Yaskawa INFORM job: tourneTRJ3.JBI

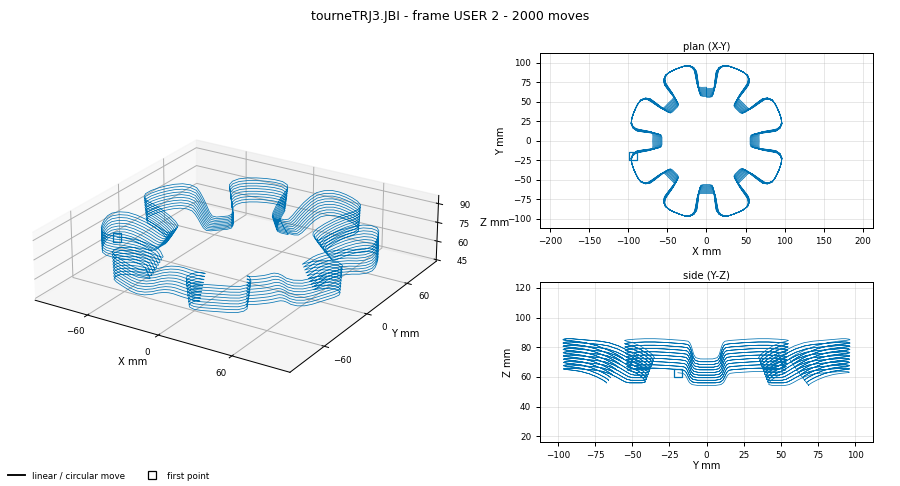
[picture p0: tool path of tourneTRJ3.JBI in frame USER 2, 2000 of 2000 moves have a stored position in this frame; points joined in program order, loops and branches not executed]
/JOB
//NAME tourneTRJ3
///FOLDERNAME DEMO
//POS
///NPOS 2000,0,2000,0,0,0
///USER 2
///TOOL 7
///POSTYPE USER
///RECTAN
///RCONF 1,0,0,0,0,0,0,0,0,0,0,0,0,0,0,0,0,0,0,0,0,0,0,0
C00000=-94.423,-19.246,62.877,176.4713,-3.4802,-10698.4794
C00001=-90.636,-15.942,62.469,177.8869,-7.7734,-10700.0243
C00002=-85.405,-14.621,61.698,179.5492,-7.9435,-10700.2854
C00003=-79.780,-13.569,60.151,179.7039,-6.1061,-10700.3475
C00004=-74.809,-12.586,58.158,179.7463,-3.0888,-10700.4499
C00005=-71.127,-11.507,56.252,-179.3006,3.5805,-10700.8103
C00006=-69.044,-9.699,54.888,-155.7698,19.6431,-10702.0037
C00007=-68.619,-6.200,54.350,-141.8645,5.1067,-10704.8371
C00008=-68.781,-2.945,54.326,-141.2129,-0.2944,-10707.5483
C00009=-68.843,0.000,54.342,-141.2230,0.0000,-10710.0000
C00010=-68.781,2.945,54.326,-141.2129,0.2944,-10712.4517
C00011=-68.619,6.200,54.350,-141.8645,-5.1067,-10715.1629
C00012=-69.044,9.699,54.888,-155.7643,-19.6439,-10717.9963
C00013=-71.127,11.507,56.252,-179.3006,-3.5805,-10719.1897
C00014=-74.809,12.586,58.158,179.7463,3.0888,-10719.5501
C00015=-79.780,13.569,60.151,179.7039,6.1061,-10719.6525
C00016=-85.405,14.621,61.698,179.5492,7.9435,-10719.7146
C00017=-90.636,15.942,62.469,177.8869,7.7734,-10719.9757
C00018=-94.423,19.246,62.877,176.4713,3.4802,-10721.5206
C00019=-96.154,24.159,63.210,177.6712,0.8456,-10724.1038
C00020=-95.429,29.718,63.547,179.8441,0.0005,-10727.2974
C00021=-93.512,35.416,63.770,179.9819,0.0007,-10730.7433
C00022=-91.166,41.080,63.770,179.9820,0.0018,-10734.2566
C00023=-88.493,46.465,63.547,179.8436,-0.0020,-10737.7026
C00024=-85.074,50.908,63.210,177.6714,-0.8446,-10740.8962
C00025=-80.376,53.158,62.877,176.4684,-3.4763,-10743.4793
C00026=-75.362,52.817,62.469,177.8861,-7.7686,-10745.0245
C00027=-70.729,50.052,61.698,179.5510,-7.9442,-10745.2855
C00028=-66.007,46.818,60.151,179.7042,-6.1110,-10745.3476
C00029=-61.798,43.998,58.158,179.7506,-3.0878,-10745.4495
C00030=-58.431,42.158,56.252,-179.3002,3.5752,-10745.8105
C00031=-55.679,41.963,54.888,-155.7662,19.6450,-10747.0038
C00032=-52.905,44.137,54.350,-141.8624,5.1087,-10749.8372
C00033=-50.718,46.553,54.326,-141.2122,-0.2913,-10752.5482
C00034=-48.679,48.679,54.342,-141.2237,-0.0052,-10755.0000
C00035=-46.553,50.718,54.326,-141.2122,0.2913,-10757.4518
C00036=-44.137,52.905,54.350,-141.8624,-5.1087,-10760.1628
C00037=-41.963,55.680,54.888,-155.7664,-19.6452,-10762.9966
C00038=-42.158,58.431,56.252,-179.3002,-3.5752,-10764.1895
C00039=-43.998,61.798,58.158,179.7506,3.0878,-10764.5505
C00040=-46.818,66.007,60.151,179.7042,6.1110,-10764.6524
C00041=-50.052,70.729,61.698,179.5510,7.9442,-10764.7145
C00042=-52.817,75.362,62.469,177.8861,7.7686,-10764.9755
C00043=-53.158,80.376,62.877,176.4684,3.4763,-10766.5207
C00044=-50.908,85.074,63.210,177.6714,0.8446,-10769.1038
C00045=-46.465,88.493,63.547,179.8436,0.0020,-10772.2974
C00046=-41.080,91.166,63.770,179.9820,-0.0018,-10775.7434
C00047=-35.416,93.512,63.770,179.9819,-0.0007,-10779.2567
C00048=-29.718,95.429,63.547,179.8441,-0.0005,-10782.7026
C00049=-24.159,96.154,63.210,177.6712,-0.8456,-10785.8962
C00050=-19.246,94.423,62.877,176.4713,-3.4802,-10788.4794
C00051=-15.942,90.636,62.469,177.8869,-7.7734,-10790.0243
C00052=-14.621,85.405,61.698,179.5492,-7.9435,-10790.2854
C00053=-13.569,79.780,60.151,179.7039,-6.1061,-10790.3475
C00054=-12.586,74.809,58.158,179.7463,-3.0888,-10790.4499
C00055=-11.507,71.127,56.252,-179.3006,3.5805,-10790.8103
C00056=-9.699,69.044,54.888,-155.7643,19.6439,-10792.0037
C00057=-6.200,68.619,54.350,-141.8645,5.1067,-10794.8371
C00058=-2.945,68.781,54.326,-141.2129,-0.2944,-10797.5483
C00059=0.000,68.843,54.342,-141.2230,-0.0000,-10800.0000
C00060=0.000,67.469,56.061,-141.5406,-0.0000,-10800.0000
C00061=2.820,67.413,56.044,-141.5283,0.3002,-10802.3954
C00062=5.989,67.263,56.069,-142.2439,-5.3506,-10805.0881
C00063=9.441,67.734,56.637,-157.1153,-19.5601,-10807.9350
C00064=11.191,69.937,58.076,-179.5522,-2.6083,-10809.0911
C00065=12.227,73.809,60.085,179.7607,3.4681,-10809.4060
C00066=13.183,79.025,62.181,179.7489,6.2113,-10809.4709
C00067=14.211,84.918,63.804,179.6316,7.9111,-10809.5004
C00068=15.500,90.396,64.610,178.0217,7.7526,-10809.7298
C00069=18.832,94.373,65.037,176.5110,3.5309,-10811.2851
C00070=23.832,96.213,65.385,177.6850,0.8573,-10813.9122
C00071=29.513,95.497,65.736,179.8387,0.0019,-10817.1736
C00072=35.347,93.539,65.969,179.9819,0.0007,-10820.7008
C00073=41.148,91.136,65.969,179.9820,0.0019,-10824.2992
C00074=46.658,88.395,65.736,179.8436,-0.0017,-10827.8267
C00075=51.181,84.885,65.385,177.6852,-0.8535,-10831.0877
C00076=53.416,80.048,65.037,176.5097,-3.5333,-10833.7152
C00077=52.959,74.880,64.610,178.0182,-7.7554,-10835.2699
C00078=49.997,70.095,63.804,179.6281,-7.9119,-10835.4993
C00079=46.557,65.200,62.181,179.7470,-6.2113,-10835.5293
C00080=43.545,60.837,60.085,179.7604,-3.4666,-10835.5938
C00081=41.540,57.367,58.076,-179.5517,2.6125,-10835.9087
C00082=41.220,54.571,56.637,-157.1158,19.5601,-10837.0654
C00083=43.327,51.796,56.069,-142.2456,5.3482,-10839.9123
C00084=45.674,49.662,56.044,-141.5313,-0.2969,-10842.6047
C00085=47.708,47.708,56.061,-141.5419,-0.0000,-10845.0000
C00086=49.662,45.674,56.044,-141.5313,0.2969,-10847.3953
C00087=51.797,43.327,56.069,-142.2457,-5.3486,-10850.0883
C00088=54.571,41.220,56.637,-157.1158,-19.5601,-10852.9346
C00089=57.367,41.540,58.076,-179.5517,-2.6125,-10854.0913
C00090=60.837,43.545,60.085,179.7604,3.4666,-10854.4062
C00091=65.200,46.557,62.181,179.7470,6.2113,-10854.4707
C00092=70.095,49.997,63.804,179.6281,7.9119,-10854.5007
C00093=74.880,52.959,64.610,178.0182,7.7554,-10854.7301
C00094=80.048,53.416,65.037,176.5097,3.5333,-10856.2848
C00095=84.885,51.181,65.385,177.6852,0.8535,-10858.9123
C00096=88.395,46.658,65.736,179.8436,0.0017,-10862.1733
C00097=91.136,41.148,65.969,179.9820,-0.0019,-10865.7008
C00098=93.539,35.347,65.969,179.9819,-0.0007,-10869.2992
C00099=95.497,29.513,65.736,179.8387,-0.0019,-10872.8264
C00100=96.213,23.832,65.385,177.6850,-0.8573,-10876.0878
C00101=94.373,18.832,65.037,176.5110,-3.5309,-10878.7149
C00102=90.396,15.500,64.610,178.0217,-7.7526,-10880.2702
C00103=84.918,14.211,63.804,179.6316,-7.9111,-10880.4996
C00104=79.025,13.183,62.181,179.7489,-6.2113,-10880.5291
C00105=73.809,12.227,60.085,179.7607,-3.4681,-10880.5940
C00106=69.937,11.191,58.076,-179.5522,2.6083,-10880.9089
C00107=67.734,9.441,56.637,-157.1153,19.5601,-10882.0650
C00108=67.263,5.989,56.069,-142.2439,5.3506,-10884.9119
C00109=67.413,2.820,56.044,-141.5283,-0.3002,-10887.6046
C00110=67.469,0.000,56.061,-141.5406,-0.0000,-10890.0000
C00111=67.413,-2.820,56.044,-141.5283,0.3002,-10892.3954
C00112=67.263,-5.989,56.069,-142.2439,-5.3506,-10895.0881
C00113=67.734,-9.441,56.637,-157.1153,-19.5601,-10897.9350
C00114=69.937,-11.191,58.076,-179.5522,-2.6083,-10899.0911
C00115=73.809,-12.227,60.085,179.7607,3.4681,-10899.4060
C00116=79.025,-13.183,62.181,179.7489,6.2113,-10899.4709
C00117=84.918,-14.211,63.804,179.6316,7.9111,-10899.5004
C00118=90.396,-15.500,64.610,178.0217,7.7526,-10899.7298
C00119=94.373,-18.832,65.037,176.5110,3.5309,-10901.2851
C00120=96.213,-23.832,65.385,177.6850,0.8573,-10903.9122
C00121=95.497,-29.513,65.736,179.8387,0.0019,-10907.1736
C00122=93.539,-35.347,65.969,179.9819,0.0007,-10910.7008
C00123=91.136,-41.148,65.969,179.9820,0.0019,-10914.2992
C00124=88.395,-46.658,65.736,179.8436,-0.0017,-10917.8267
C00125=84.885,-51.181,65.385,177.6852,-0.8535,-10921.0877
C00126=80.048,-53.416,65.037,176.5097,-3.5333,-10923.7152
C00127=74.880,-52.959,64.610,178.0182,-7.7554,-10925.2699
C00128=70.095,-49.997,63.804,179.6281,-7.9119,-10925.4993
C00129=65.200,-46.557,62.181,179.7470,-6.2113,-10925.5293
C00130=60.837,-43.545,60.085,179.7604,-3.4666,-10925.5938
C00131=57.367,-41.540,58.076,-179.5517,2.6125,-10925.9087
C00132=54.571,-41.220,56.637,-157.1158,19.5601,-10927.0654
C00133=51.796,-43.327,56.069,-142.2456,5.3482,-10929.9123
C00134=49.662,-45.674,56.044,-141.5313,-0.2969,-10932.6047
C00135=47.708,-47.708,56.061,-141.5419,0.0000,-10935.0000
C00136=45.674,-49.662,56.044,-141.5313,0.2969,-10937.3953
C00137=43.327,-51.797,56.069,-142.2457,-5.3486,-10940.0883
C00138=41.220,-54.571,56.637,-157.1158,-19.5601,-10942.9346
C00139=41.540,-57.367,58.076,-179.5517,-2.6125,-10944.0913
C00140=43.545,-60.837,60.085,179.7604,3.4666,-10944.4062
C00141=46.557,-65.200,62.181,179.7470,6.2113,-10944.4707
C00142=49.997,-70.095,63.804,179.6281,7.9119,-10944.5007
C00143=52.959,-74.880,64.610,178.0182,7.7554,-10944.7301
C00144=53.416,-80.048,65.037,176.5097,3.5333,-10946.2848
C00145=51.181,-84.885,65.385,177.6852,0.8535,-10948.9123
C00146=46.658,-88.395,65.736,179.8436,0.0017,-10952.1733
C00147=41.148,-91.136,65.969,179.9820,-0.0019,-10955.7008
C00148=35.347,-93.539,65.969,179.9819,-0.0007,-10959.2992
C00149=29.513,-95.497,65.736,179.8387,-0.0019,-10962.8264
C00150=23.832,-96.213,65.385,177.6850,-0.8573,-10966.0878
C00151=18.832,-94.373,65.037,176.5110,-3.5309,-10968.7149
C00152=15.500,-90.396,64.610,178.0217,-7.7526,-10970.2702
C00153=14.211,-84.918,63.804,179.6316,-7.9111,-10970.4996
C00154=13.183,-79.025,62.181,179.7489,-6.2113,-10970.5291
C00155=12.227,-73.809,60.085,179.7607,-3.4681,-10970.5940
C00156=11.191,-69.937,58.076,-179.5522,2.6083,-10970.9089
C00157=9.441,-67.734,56.637,-157.1153,19.5601,-10972.0650
C00158=5.989,-67.263,56.069,-142.2439,5.3506,-10974.9119
C00159=2.820,-67.413,56.044,-141.5283,-0.3002,-10977.6046
C00160=0.000,-67.469,56.061,-141.5406,0.0000,-10980.0000
C00161=0.000,-67.469,56.061,-141.5406,0.0000,-10980.0000
C00162=-2.820,-67.413,56.044,-141.5283,0.3002,-10982.3954
C00163=-5.989,-67.263,56.069,-142.2439,-5.3506,-10985.0881
C00164=-9.441,-67.734,56.637,-157.1153,-19.5601,-10987.9350
C00165=-11.191,-69.937,58.076,-179.5522,-2.6083,-10989.0911
C00166=-12.227,-73.809,60.085,179.7607,3.4681,-10989.4060
C00167=-13.183,-79.025,62.181,179.7489,6.2113,-10989.4709
C00168=-14.211,-84.918,63.804,179.6316,7.9111,-10989.5004
C00169=-15.500,-90.396,64.610,178.0217,7.7526,-10989.7298
C00170=-18.832,-94.373,65.037,176.5110,3.5309,-10991.2851
C00171=-23.832,-96.213,65.385,177.6850,0.8573,-10993.9122
C00172=-29.513,-95.497,65.736,179.8387,0.0019,-10997.1736
C00173=-35.347,-93.539,65.969,179.9819,0.0007,-11000.7008
C00174=-41.148,-91.136,65.969,179.9820,0.0019,-11004.2992
C00175=-46.658,-88.395,65.736,179.8436,-0.0017,-11007.8267
C00176=-51.181,-84.885,65.385,177.6852,-0.8535,-11011.0877
C00177=-53.416,-80.048,65.037,176.5097,-3.5333,-11013.7152
C00178=-52.959,-74.880,64.610,178.0182,-7.7554,-11015.2699
C00179=-49.997,-70.095,63.804,179.6281,-7.9119,-11015.4993
C00180=-46.557,-65.200,62.181,179.7470,-6.2113,-11015.5293
C00181=-43.545,-60.837,60.085,179.7604,-3.4666,-11015.5938
C00182=-41.540,-57.367,58.076,-179.5517,2.6125,-11015.9087
C00183=-41.220,-54.571,56.637,-157.1158,19.5601,-11017.0654
C00184=-43.327,-51.796,56.069,-142.2456,5.3482,-11019.9123
C00185=-45.674,-49.662,56.044,-141.5313,-0.2969,-11022.6047
C00186=-47.708,-47.708,56.061,-141.5419,0.0000,-11025.0000
C00187=-49.662,-45.674,56.044,-141.5313,0.2969,-11027.3953
C00188=-51.797,-43.327,56.069,-142.2457,-5.3486,-11030.0883
C00189=-54.571,-41.220,56.637,-157.1158,-19.5601,-11032.9346
C00190=-57.367,-41.540,58.076,-179.5517,-2.6125,-11034.0913
C00191=-60.837,-43.545,60.085,179.7604,3.4666,-11034.4062
C00192=-65.200,-46.557,62.181,179.7470,6.2113,-11034.4707
C00193=-70.095,-49.997,63.804,179.6281,7.9119,-11034.5007
C00194=-74.880,-52.959,64.610,178.0182,7.7554,-11034.7301
C00195=-80.048,-53.416,65.037,176.5097,3.5333,-11036.2848
C00196=-84.885,-51.181,65.385,177.6852,0.8535,-11038.9123
C00197=-88.395,-46.658,65.736,179.8436,0.0017,-11042.1733
C00198=-91.136,-41.148,65.969,179.9820,-0.0019,-11045.7008
C00199=-93.539,-35.347,65.969,179.9819,-0.0007,-11049.2992
C00200=-95.497,-29.513,65.736,179.8387,-0.0019,-11052.8264
C00201=-96.213,-23.832,65.385,177.6850,-0.8573,-11056.0878
C00202=-94.373,-18.832,65.037,176.5110,-3.5309,-11058.7149
C00203=-90.396,-15.500,64.610,178.0217,-7.7526,-11060.2702
C00204=-84.918,-14.211,63.804,179.6316,-7.9111,-11060.4996
C00205=-79.025,-13.183,62.181,179.7489,-6.2113,-11060.5291
C00206=-73.809,-12.227,60.085,179.7607,-3.4681,-11060.5940
C00207=-69.937,-11.191,58.076,-179.5522,2.6083,-11060.9089
C00208=-67.734,-9.441,56.637,-157.1153,19.5601,-11062.0650
C00209=-67.263,-5.989,56.069,-142.2439,5.3506,-11064.9119
C00210=-67.413,-2.820,56.044,-141.5283,-0.3002,-11067.6046
C00211=-67.469,0.000,56.061,-141.5406,0.0000,-11070.0000
C00212=-67.413,2.820,56.044,-141.5283,0.3002,-11072.3954
C00213=-67.263,5.989,56.069,-142.2439,-5.3506,-11075.0881
C00214=-67.734,9.441,56.637,-157.1153,-19.5601,-11077.9350
C00215=-69.937,11.191,58.076,-179.5522,-2.6083,-11079.0911
C00216=-73.809,12.227,60.085,179.7607,3.4681,-11079.4060
C00217=-79.025,13.183,62.181,179.7489,6.2113,-11079.4709
C00218=-84.918,14.211,63.804,179.6316,7.9111,-11079.5004
C00219=-90.396,15.500,64.610,178.0217,7.7526,-11079.7298
C00220=-94.373,18.832,65.037,176.5110,3.5309,-11081.2851
C00221=-96.213,23.832,65.385,177.6850,0.8573,-11083.9122
C00222=-95.497,29.513,65.736,179.8387,0.0019,-11087.1736
C00223=-93.539,35.347,65.969,179.9819,0.0007,-11090.7008
C00224=-91.136,41.148,65.969,179.9820,0.0019,-11094.2992
C00225=-88.395,46.658,65.736,179.8436,-0.0017,-11097.8267
C00226=-84.885,51.181,65.385,177.6852,-0.8535,-11101.0877
C00227=-80.048,53.416,65.037,176.5097,-3.5333,-11103.7152
C00228=-74.880,52.959,64.610,178.0182,-7.7554,-11105.2699
C00229=-70.095,49.997,63.804,179.6281,-7.9119,-11105.4993
C00230=-65.200,46.557,62.181,179.7470,-6.2113,-11105.5293
C00231=-60.837,43.545,60.085,179.7604,-3.4666,-11105.5938
C00232=-57.367,41.540,58.076,-179.5517,2.6125,-11105.9087
C00233=-54.571,41.220,56.637,-157.1158,19.5601,-11107.0654
C00234=-51.796,43.327,56.069,-142.2456,5.3482,-11109.9123
C00235=-49.662,45.674,56.044,-141.5313,-0.2969,-11112.6047
C00236=-47.708,47.708,56.061,-141.5419,0.0000,-11115.0000
C00237=-45.674,49.662,56.044,-141.5313,0.2969,-11117.3953
C00238=-43.327,51.797,56.069,-142.2457,-5.3486,-11120.0883
C00239=-41.220,54.571,56.637,-157.1158,-19.5601,-11122.9346
C00240=-41.540,57.367,58.076,-179.5517,-2.6125,-11124.0913
C00241=-43.545,60.837,60.085,179.7604,3.4666,-11124.4062
C00242=-46.557,65.200,62.181,179.7470,6.2113,-11124.4707
C00243=-49.997,70.095,63.804,179.6281,7.9119,-11124.5007
C00244=-52.959,74.880,64.610,178.0182,7.7554,-11124.7301
C00245=-53.416,80.048,65.037,176.5097,3.5333,-11126.2848
C00246=-51.181,84.885,65.385,177.6852,0.8535,-11128.9123
C00247=-46.658,88.395,65.736,179.8436,0.0017,-11132.1733
C00248=-41.148,91.136,65.969,179.9820,-0.0019,-11135.7008
C00249=-35.347,93.539,65.969,179.9819,-0.0007,-11139.2992
C00250=-29.513,95.497,65.736,179.8387,-0.0019,-11142.8264
C00251=-23.832,96.213,65.385,177.6850,-0.8573,-11146.0878
C00252=-18.832,94.373,65.037,176.5110,-3.5309,-11148.7149
C00253=-15.500,90.396,64.610,178.0217,-7.7526,-11150.2702
C00254=-14.211,84.918,63.804,179.6316,-7.9111,-11150.4996
C00255=-13.183,79.025,62.181,179.7489,-6.2113,-11150.5291
C00256=-12.227,73.809,60.085,179.7607,-3.4681,-11150.5940
C00257=-11.191,69.937,58.076,-179.5522,2.6083,-11150.9089
C00258=-9.441,67.734,56.637,-157.1153,19.5601,-11152.0650
C00259=-5.989,67.263,56.069,-142.2439,5.3506,-11154.9119
C00260=-2.820,67.413,56.044,-141.5283,-0.3002,-11157.6046
C00261=0.000,67.469,56.061,-141.5406,0.0000,-11160.0000
C00262=0.000,66.107,57.788,-141.9406,0.0000,-11160.0000
C00263=2.695,66.055,57.771,-141.9333,0.3033,-11162.3363
C00264=5.779,65.917,57.797,-142.7097,-5.5769,-11165.0104
C00265=9.185,66.436,58.394,-158.5027,-19.3588,-11167.8714
C00266=10.880,68.762,59.909,-179.7398,-1.7295,-11168.9912
C00267=11.874,72.826,62.021,179.7781,3.7717,-11169.2604
C00268=12.805,78.288,64.219,179.7878,6.2471,-11169.2892
C00269=13.814,84.445,65.915,179.6969,7.8067,-11169.2905
C00270=15.073,90.163,66.756,178.1578,7.6627,-11169.4907
C00271=18.432,94.325,67.200,176.5834,3.5410,-11171.0568
C00272=23.517,96.271,67.561,177.7197,0.8583,-11173.7273
C00273=29.315,95.562,67.927,179.8441,-0.0001,-11177.0541
C00274=35.280,93.564,68.167,179.9819,0.0007,-11180.6599
C00275=41.213,91.107,68.167,179.9820,0.0019,-11184.3400
C00276=46.844,88.301,67.927,179.8436,-0.0014,-11187.9461
C00277=51.445,84.703,67.561,177.7227,-0.8571,-11191.2727
C00278=53.664,79.731,67.200,176.5830,-3.5436,-11193.9430
C00279=53.097,74.413,66.756,178.1541,-7.6603,-11195.5096
C00280=49.944,69.479,65.915,179.6940,-7.8083,-11195.7099
C00281=46.303,64.413,64.219,179.7915,-6.2491,-11195.7103
C00282=43.100,59.892,62.021,179.7771,-3.7746,-11195.7399
C00283=40.929,56.315,59.909,-179.7405,1.7313,-11196.0092
C00284=40.483,53.472,58.394,-158.5003,19.3574,-11197.1289
C00285=42.524,50.697,57.797,-142.7113,5.5764,-11199.9895
C00286=44.802,48.614,57.771,-141.9338,-0.3012,-11202.6632
C00287=46.745,46.745,57.788,-141.9426,0.0000,-11205.0000
C00288=48.613,44.802,57.771,-141.9338,0.3016,-11207.3362
C00289=50.697,42.524,57.797,-142.7148,-5.5810,-11210.0105
C00290=53.472,40.483,58.395,-158.5003,-19.3574,-11212.8711
C00291=56.315,40.929,59.909,-179.7405,-1.7313,-11213.9908
C00292=59.892,43.100,62.021,179.7771,3.7746,-11214.2601
C00293=64.413,46.303,64.219,179.7915,6.2491,-11214.2897
C00294=69.479,49.944,65.915,179.6940,7.8083,-11214.2901
C00295=74.413,53.097,66.756,178.1541,7.6603,-11214.4904
C00296=79.731,53.664,67.200,176.5830,3.5436,-11216.0570
C00297=84.703,51.445,67.561,177.7227,0.8571,-11218.7273
C00298=88.301,46.844,67.927,179.8436,0.0014,-11222.0539
C00299=91.107,41.213,68.167,179.9820,-0.0019,-11225.6600
C00300=93.564,35.280,68.167,179.9819,-0.0007,-11229.3401
C00301=95.562,29.315,67.927,179.8441,0.0001,-11232.9459
C00302=96.271,23.517,67.561,177.7197,-0.8583,-11236.2727
C00303=94.325,18.432,67.200,176.5834,-3.5410,-11238.9432
C00304=90.163,15.073,66.756,178.1578,-7.6627,-11240.5093
C00305=84.445,13.814,65.915,179.6969,-7.8067,-11240.7095
C00306=78.288,12.805,64.219,179.7878,-6.2471,-11240.7108
C00307=72.826,11.874,62.021,179.7781,-3.7717,-11240.7396
C00308=68.762,10.880,59.909,-179.7398,1.7295,-11241.0088
C00309=66.436,9.185,58.394,-158.5027,19.3588,-11242.1286
C00310=65.917,5.779,57.797,-142.7097,5.5769,-11244.9896
C00311=66.055,2.695,57.771,-141.9333,-0.3033,-11247.6637
C00312=66.107,0.000,57.788,-141.9406,-0.0000,-11250.0000
C00313=66.055,-2.695,57.771,-141.9333,0.3033,-11252.3363
C00314=65.917,-5.780,57.797,-142.7102,-5.5846,-11255.0112
C00315=66.436,-9.185,58.395,-158.5027,-19.3588,-11257.8714
C00316=68.762,-10.880,59.909,-179.7398,-1.7295,-11258.9912
C00317=72.826,-11.874,62.021,179.7781,3.7717,-11259.2604
C00318=78.288,-12.805,64.219,179.7878,6.2471,-11259.2892
C00319=84.445,-13.814,65.915,179.6969,7.8067,-11259.2905
C00320=90.163,-15.073,66.756,178.1578,7.6627,-11259.4907
C00321=94.325,-18.432,67.200,176.5834,3.5410,-11261.0568
C00322=96.271,-23.517,67.561,177.7197,0.8583,-11263.7273
C00323=95.562,-29.315,67.927,179.8441,-0.0001,-11267.0541
C00324=93.564,-35.280,68.167,179.9819,0.0007,-11270.6599
C00325=91.107,-41.213,68.167,179.9820,0.0019,-11274.3400
C00326=88.301,-46.844,67.927,179.8436,-0.0014,-11277.9461
C00327=84.703,-51.445,67.561,177.7227,-0.8571,-11281.2727
C00328=79.731,-53.664,67.200,176.5830,-3.5436,-11283.9430
C00329=74.413,-53.097,66.756,178.1541,-7.6603,-11285.5096
C00330=69.479,-49.944,65.915,179.6940,-7.8083,-11285.7099
C00331=64.413,-46.303,64.219,179.7915,-6.2491,-11285.7103
C00332=59.892,-43.100,62.021,179.7771,-3.7746,-11285.7399
C00333=56.315,-40.929,59.909,-179.7405,1.7313,-11286.0092
C00334=53.472,-40.483,58.394,-158.5003,19.3574,-11287.1289
C00335=50.697,-42.524,57.797,-142.7113,5.5764,-11289.9895
C00336=48.614,-44.802,57.771,-141.9338,-0.3012,-11292.6632
C00337=46.745,-46.745,57.788,-141.9426,-0.0000,-11295.0000
C00338=44.802,-48.613,57.771,-141.9338,0.3016,-11297.3362
C00339=42.524,-50.697,57.797,-142.7148,-5.5810,-11300.0105
C00340=40.483,-53.472,58.395,-158.5003,-19.3574,-11302.8711
C00341=40.929,-56.315,59.909,-179.7405,-1.7313,-11303.9908
C00342=43.100,-59.892,62.021,179.7771,3.7746,-11304.2601
C00343=46.303,-64.413,64.219,179.7915,6.2491,-11304.2897
C00344=49.944,-69.479,65.915,179.6940,7.8083,-11304.2901
C00345=53.097,-74.413,66.756,178.1541,7.6603,-11304.4904
C00346=53.664,-79.731,67.200,176.5830,3.5436,-11306.0570
C00347=51.445,-84.703,67.561,177.7227,0.8571,-11308.7273
C00348=46.844,-88.301,67.927,179.8436,0.0014,-11312.0539
C00349=41.213,-91.107,68.167,179.9820,-0.0019,-11315.6600
C00350=35.280,-93.564,68.167,179.9819,-0.0007,-11319.3401
C00351=29.315,-95.562,67.927,179.8441,0.0001,-11322.9459
C00352=23.517,-96.271,67.561,177.7197,-0.8583,-11326.2727
C00353=18.432,-94.325,67.200,176.5834,-3.5410,-11328.9432
C00354=15.073,-90.163,66.756,178.1578,-7.6627,-11330.5093
C00355=13.814,-84.445,65.915,179.6969,-7.8067,-11330.7095
C00356=12.805,-78.288,64.219,179.7878,-6.2471,-11330.7108
C00357=11.874,-72.826,62.021,179.7781,-3.7717,-11330.7396
C00358=10.880,-68.762,59.909,-179.7398,1.7295,-11331.0088
C00359=9.185,-66.436,58.394,-158.5027,19.3588,-11332.1286
C00360=5.779,-65.917,57.797,-142.7097,5.5769,-11334.9896
C00361=2.695,-66.055,57.771,-141.9333,-0.3033,-11337.6637
C00362=0.000,-66.107,57.788,-141.9406,-0.0000,-11340.0000
C00363=0.000,-66.107,57.788,-141.9406,-0.0000,-11340.0000
C00364=-2.695,-66.055,57.771,-141.9333,0.3033,-11342.3363
C00365=-5.780,-65.917,57.797,-142.7102,-5.5846,-11345.0112
C00366=-9.185,-66.436,58.395,-158.5027,-19.3588,-11347.8714
C00367=-10.880,-68.762,59.909,-179.7398,-1.7295,-11348.9912
C00368=-11.874,-72.826,62.021,179.7781,3.7717,-11349.2604
C00369=-12.805,-78.288,64.219,179.7878,6.2471,-11349.2892
C00370=-13.814,-84.445,65.915,179.6969,7.8067,-11349.2905
C00371=-15.073,-90.163,66.756,178.1578,7.6627,-11349.4907
C00372=-18.432,-94.325,67.200,176.5834,3.5410,-11351.0568
C00373=-23.517,-96.271,67.561,177.7197,0.8583,-11353.7273
C00374=-29.315,-95.562,67.927,179.8441,-0.0001,-11357.0541
C00375=-35.280,-93.564,68.167,179.9819,0.0007,-11360.6599
C00376=-41.213,-91.107,68.167,179.9820,0.0019,-11364.3400
C00377=-46.844,-88.301,67.927,179.8436,-0.0014,-11367.9461
C00378=-51.445,-84.703,67.561,177.7227,-0.8571,-11371.2727
C00379=-53.664,-79.731,67.200,176.5830,-3.5436,-11373.9430
C00380=-53.097,-74.413,66.756,178.1541,-7.6603,-11375.5096
C00381=-49.944,-69.479,65.915,179.6940,-7.8083,-11375.7099
C00382=-46.303,-64.413,64.219,179.7915,-6.2491,-11375.7103
C00383=-43.100,-59.892,62.021,179.7771,-3.7746,-11375.7399
C00384=-40.929,-56.315,59.909,-179.7405,1.7313,-11376.0092
C00385=-40.483,-53.472,58.394,-158.5003,19.3574,-11377.1289
C00386=-42.524,-50.697,57.797,-142.7113,5.5764,-11379.9895
C00387=-44.802,-48.614,57.771,-141.9338,-0.3012,-11382.6632
C00388=-46.745,-46.745,57.788,-141.9426,-0.0000,-11385.0000
C00389=-48.613,-44.802,57.771,-141.9338,0.3016,-11387.3362
C00390=-50.697,-42.524,57.797,-142.7148,-5.5810,-11390.0105
C00391=-53.472,-40.483,58.395,-158.5003,-19.3574,-11392.8711
C00392=-56.315,-40.929,59.909,-179.7405,-1.7313,-11393.9908
C00393=-59.892,-43.100,62.021,179.7771,3.7746,-11394.2601
C00394=-64.413,-46.303,64.219,179.7915,6.2491,-11394.2897
C00395=-69.479,-49.944,65.915,179.6940,7.8083,-11394.2901
C00396=-74.413,-53.097,66.756,178.1541,7.6603,-11394.4904
C00397=-79.731,-53.664,67.200,176.5830,3.5436,-11396.0570
C00398=-84.703,-51.445,67.561,177.7227,0.8571,-11398.7273
C00399=-88.301,-46.844,67.927,179.8436,0.0014,-11402.0539
C00400=-91.107,-41.213,68.167,179.9820,-0.0019,-11405.6600
C00401=-93.564,-35.280,68.167,179.9819,-0.0007,-11409.3401
C00402=-95.562,-29.315,67.927,179.8441,0.0001,-11412.9459
C00403=-96.271,-23.517,67.561,177.7197,-0.8583,-11416.2727
C00404=-94.325,-18.432,67.200,176.5834,-3.5410,-11418.9432
C00405=-90.163,-15.073,66.756,178.1578,-7.6627,-11420.5093
C00406=-84.445,-13.814,65.915,179.6969,-7.8067,-11420.7095
C00407=-78.288,-12.805,64.219,179.7878,-6.2471,-11420.7108
C00408=-72.826,-11.874,62.021,179.7781,-3.7717,-11420.7396
C00409=-68.762,-10.880,59.909,-179.7398,1.7295,-11421.0088
C00410=-66.436,-9.185,58.394,-158.5027,19.3588,-11422.1286
C00411=-65.917,-5.779,57.797,-142.7097,5.5769,-11424.9896
C00412=-66.055,-2.695,57.771,-141.9333,-0.3033,-11427.6637
C00413=-66.107,0.000,57.788,-141.9406,0.0000,-11430.0000
C00414=-66.055,2.695,57.771,-141.9333,0.3033,-11432.3363
C00415=-65.917,5.780,57.797,-142.7102,-5.5846,-11435.0112
C00416=-66.436,9.185,58.395,-158.5027,-19.3588,-11437.8714
C00417=-68.762,10.880,59.909,-179.7398,-1.7295,-11438.9912
C00418=-72.826,11.874,62.021,179.7781,3.7717,-11439.2604
C00419=-78.288,12.805,64.219,179.7878,6.2471,-11439.2892
C00420=-84.445,13.814,65.915,179.6969,7.8067,-11439.2905
C00421=-90.163,15.073,66.756,178.1578,7.6627,-11439.4907
C00422=-94.325,18.432,67.200,176.5834,3.5410,-11441.0568
C00423=-96.271,23.517,67.561,177.7197,0.8583,-11443.7273
C00424=-95.562,29.315,67.927,179.8441,-0.0001,-11447.0541
C00425=-93.564,35.280,68.167,179.9819,0.0007,-11450.6599
C00426=-91.107,41.213,68.167,179.9820,0.0019,-11454.3400
C00427=-88.301,46.844,67.927,179.8436,-0.0014,-11457.9461
C00428=-84.703,51.445,67.561,177.7227,-0.8571,-11461.2727
C00429=-79.731,53.664,67.200,176.5830,-3.5436,-11463.9430
C00430=-74.413,53.097,66.756,178.1541,-7.6603,-11465.5096
C00431=-69.479,49.944,65.915,179.6940,-7.8083,-11465.7099
C00432=-64.413,46.303,64.219,179.7915,-6.2491,-11465.7103
C00433=-59.892,43.100,62.021,179.7771,-3.7746,-11465.7399
C00434=-56.315,40.929,59.909,-179.7405,1.7313,-11466.0092
C00435=-53.472,40.483,58.394,-158.5003,19.3574,-11467.1289
C00436=-50.697,42.524,57.797,-142.7113,5.5764,-11469.9895
C00437=-48.614,44.802,57.771,-141.9338,-0.3012,-11472.6632
C00438=-46.745,46.745,57.788,-141.9426,0.0000,-11475.0000
C00439=-44.802,48.613,57.771,-141.9338,0.3016,-11477.3362
C00440=-42.524,50.697,57.797,-142.7148,-5.5810,-11480.0105
C00441=-40.483,53.472,58.395,-158.5003,-19.3574,-11482.8711
C00442=-40.929,56.315,59.909,-179.7405,-1.7313,-11483.9908
C00443=-43.100,59.892,62.021,179.7771,3.7746,-11484.2601
C00444=-46.303,64.413,64.219,179.7915,6.2491,-11484.2897
C00445=-49.944,69.479,65.915,179.6940,7.8083,-11484.2901
C00446=-53.097,74.413,66.756,178.1541,7.6603,-11484.4904
C00447=-53.664,79.731,67.200,176.5830,3.5436,-11486.0570
C00448=-51.445,84.703,67.561,177.7227,0.8571,-11488.7273
C00449=-46.844,88.301,67.927,179.8436,0.0014,-11492.0539
C00450=-41.213,91.107,68.167,179.9820,-0.0019,-11495.6600
C00451=-35.280,93.564,68.167,179.9819,-0.0007,-11499.3401
C00452=-29.315,95.562,67.927,179.8441,0.0001,-11502.9459
C00453=-23.517,96.271,67.561,177.7197,-0.8583,-11506.2727
C00454=-18.432,94.325,67.200,176.5834,-3.5410,-11508.9432
C00455=-15.073,90.163,66.756,178.1578,-7.6627,-11510.5093
C00456=-13.814,84.445,65.915,179.6969,-7.8067,-11510.7095
C00457=-12.805,78.288,64.219,179.7878,-6.2471,-11510.7108
C00458=-11.874,72.826,62.021,179.7781,-3.7717,-11510.7396
C00459=-10.880,68.762,59.909,-179.7398,1.7295,-11511.0088
C00460=-9.185,66.436,58.395,-158.5027,19.3588,-11512.1286
C00461=-5.780,65.917,57.797,-142.7102,5.5846,-11514.9888
C00462=-2.695,66.055,57.771,-141.9333,-0.3033,-11517.6637
C00463=0.000,66.107,57.788,-141.9406,0.0000,-11520.0000
C00464=0.000,64.758,59.526,-142.4265,0.0000,-11520.0000
C00465=2.572,64.710,59.508,-142.4163,0.3021,-11522.2761
C00466=5.572,64.584,59.535,-143.2704,-5.7854,-11524.9310
C00467=8.932,65.152,60.163,-159.9092,-19.0297,-11527.8063
C00468=10.572,67.603,61.754,-179.8747,-0.9417,-11528.8881
C00469=11.527,71.864,63.969,179.8008,4.0103,-11529.1126
C00470=12.439,77.571,66.266,179.8289,6.2253,-11529.1102
C00471=13.430,83.988,68.033,179.7593,7.6388,-11529.0849
C00472=14.662,89.940,68.906,178.2885,7.4940,-11529.2589
C00473=18.048,94.279,69.366,176.6898,3.5102,-11530.8371
C00474=23.215,96.325,69.740,177.7754,0.8490,-11533.5503
C00475=29.126,95.625,70.117,179.8441,-0.0004,-11536.9400
C00476=35.216,93.589,70.366,179.9819,0.0007,-11540.6205
C00477=41.276,91.079,70.366,179.9820,0.0019,-11544.3795
C00478=47.022,88.212,70.117,179.8436,-0.0010,-11548.0601
C00479=51.697,84.528,69.740,177.7771,-0.8446,-11551.4498
C00480=53.903,79.427,69.366,176.6864,-3.5117,-11554.1627
C00481=53.229,73.964,68.906,178.2928,-7.4966,-11555.7411
C00482=49.892,68.885,68.033,179.7592,-7.6390,-11555.9150
C00483=46.056,63.647,66.266,179.8302,-6.2269,-11555.8901
C00484=42.664,58.966,63.969,179.7966,-4.0079,-11555.8871
C00485=40.327,55.279,61.754,-179.8773,0.9460,-11556.1114
C00486=39.754,52.385,60.163,-159.9107,19.0306,-11557.1942
C00487=41.728,49.608,59.535,-143.2689,5.7817,-11560.0690
C00488=43.938,47.576,59.508,-142.4189,-0.3039,-11562.7235
C00489=45.791,45.791,59.526,-142.4261,0.0000,-11565.0000
C00490=47.575,43.938,59.508,-142.4189,0.3043,-11567.2759
C00491=49.608,41.728,59.535,-143.2694,-5.7917,-11569.9310
C00492=52.385,39.754,60.163,-159.9107,-19.0306,-11572.8058
C00493=55.279,40.327,61.754,-179.8773,-0.9460,-11573.8886
C00494=58.966,42.664,63.969,179.7966,4.0079,-11574.1129
C00495=63.647,46.056,66.266,179.8302,6.2269,-11574.1099
C00496=68.885,49.892,68.033,179.7592,7.6390,-11574.0850
C00497=73.964,53.229,68.906,178.2928,7.4966,-11574.2589
C00498=79.427,53.903,69.366,176.6864,3.5117,-11575.8373
C00499=84.528,51.697,69.740,177.7771,0.8446,-11578.5502
C00500=88.212,47.022,70.117,179.8436,0.0010,-11581.9399
C00501=91.079,41.276,70.366,179.9820,-0.0019,-11585.6205
C00502=93.589,35.216,70.366,179.9819,-0.0007,-11589.3795
C00503=95.625,29.126,70.117,179.8441,0.0004,-11593.0600
C00504=96.325,23.215,69.740,177.7754,-0.8490,-11596.4497
C00505=94.279,18.048,69.366,176.6898,-3.5102,-11599.1629
C00506=89.940,14.662,68.906,178.2885,-7.4940,-11600.7411
C00507=83.988,13.430,68.033,179.7593,-7.6388,-11600.9151
C00508=77.571,12.439,66.266,179.8289,-6.2253,-11600.8898
C00509=71.864,11.527,63.969,179.8008,-4.0103,-11600.8874
C00510=67.603,10.572,61.754,-179.8747,0.9417,-11601.1119
C00511=65.152,8.932,60.163,-159.9092,19.0297,-11602.1937
C00512=64.584,5.572,59.535,-143.2704,5.7854,-11605.0690
C00513=64.710,2.572,59.508,-142.4163,-0.3021,-11607.7239
C00514=64.758,0.000,59.526,-142.4265,0.0000,-11610.0000
C00515=64.710,-2.572,59.508,-142.4163,0.3021,-11612.2761
C00516=64.584,-5.572,59.535,-143.2704,-5.7854,-11614.9310
C00517=65.152,-8.932,60.163,-159.9092,-19.0297,-11617.8063
C00518=67.603,-10.572,61.754,-179.8747,-0.9417,-11618.8881
C00519=71.864,-11.527,63.969,179.8008,4.0103,-11619.1126
C00520=77.571,-12.439,66.266,179.8289,6.2253,-11619.1102
C00521=83.988,-13.430,68.033,179.7593,7.6388,-11619.0849
C00522=89.940,-14.662,68.906,178.2885,7.4940,-11619.2589
C00523=94.279,-18.048,69.366,176.6898,3.5102,-11620.8371
C00524=96.325,-23.215,69.740,177.7754,0.8490,-11623.5503
C00525=95.625,-29.126,70.117,179.8441,-0.0004,-11626.9400
C00526=93.589,-35.216,70.366,179.9819,0.0007,-11630.6205
C00527=91.079,-41.276,70.366,179.9820,0.0019,-11634.3795
C00528=88.212,-47.022,70.117,179.8436,-0.0010,-11638.0601
C00529=84.528,-51.697,69.740,177.7771,-0.8446,-11641.4498
C00530=79.427,-53.903,69.366,176.6864,-3.5117,-11644.1627
C00531=73.964,-53.229,68.906,178.2928,-7.4966,-11645.7411
C00532=68.885,-49.892,68.033,179.7592,-7.6390,-11645.9150
C00533=63.647,-46.056,66.266,179.8302,-6.2269,-11645.8901
C00534=58.966,-42.664,63.969,179.7966,-4.0079,-11645.8871
C00535=55.279,-40.327,61.754,-179.8773,0.9460,-11646.1114
C00536=52.385,-39.754,60.163,-159.9107,19.0306,-11647.1942
C00537=49.608,-41.728,59.535,-143.2689,5.7817,-11650.0690
C00538=47.576,-43.938,59.508,-142.4189,-0.3039,-11652.7235
C00539=45.791,-45.791,59.526,-142.4261,0.0000,-11655.0000
C00540=43.938,-47.575,59.508,-142.4189,0.3043,-11657.2759
C00541=41.728,-49.608,59.535,-143.2694,-5.7917,-11659.9310
C00542=39.754,-52.385,60.163,-159.9107,-19.0306,-11662.8058
C00543=40.327,-55.279,61.754,-179.8773,-0.9460,-11663.8886
C00544=42.664,-58.966,63.969,179.7966,4.0079,-11664.1129
C00545=46.056,-63.647,66.266,179.8302,6.2269,-11664.1099
C00546=49.892,-68.885,68.033,179.7592,7.6390,-11664.0850
C00547=53.229,-73.964,68.906,178.2928,7.4966,-11664.2589
C00548=53.903,-79.427,69.366,176.6864,3.5117,-11665.8373
C00549=51.697,-84.528,69.740,177.7771,0.8446,-11668.5502
C00550=47.022,-88.212,70.117,179.8436,0.0010,-11671.9399
C00551=41.276,-91.079,70.366,179.9820,-0.0019,-11675.6205
C00552=35.216,-93.589,70.366,179.9819,-0.0007,-11679.3795
C00553=29.126,-95.625,70.117,179.8441,0.0004,-11683.0600
C00554=23.215,-96.325,69.740,177.7754,-0.8490,-11686.4497
C00555=18.048,-94.279,69.366,176.6898,-3.5102,-11689.1629
C00556=14.662,-89.940,68.906,178.2885,-7.4940,-11690.7411
C00557=13.430,-83.988,68.033,179.7593,-7.6388,-11690.9151
C00558=12.439,-77.571,66.266,179.8289,-6.2253,-11690.8898
C00559=11.527,-71.864,63.969,179.8008,-4.0103,-11690.8874
C00560=10.572,-67.603,61.754,-179.8747,0.9417,-11691.1119
C00561=8.932,-65.152,60.163,-159.9092,19.0297,-11692.1937
C00562=5.572,-64.584,59.535,-143.2704,5.7854,-11695.0690
C00563=2.572,-64.710,59.508,-142.4163,-0.3021,-11697.7239
C00564=0.000,-64.758,59.526,-142.4265,-0.0000,-11700.0000
C00565=0.000,-64.758,59.526,-142.4265,-0.0000,-11700.0000
C00566=-2.572,-64.710,59.508,-142.4163,0.3021,-11702.2761
C00567=-5.572,-64.584,59.535,-143.2704,-5.7854,-11704.9310
C00568=-8.932,-65.152,60.163,-159.9092,-19.0297,-11707.8063
C00569=-10.572,-67.603,61.754,-179.8747,-0.9417,-11708.8881
C00570=-11.527,-71.864,63.969,179.8008,4.0103,-11709.1126
C00571=-12.439,-77.571,66.266,179.8289,6.2253,-11709.1102
C00572=-13.430,-83.988,68.033,179.7593,7.6388,-11709.0849
C00573=-14.662,-89.940,68.906,178.2885,7.4940,-11709.2589
C00574=-18.048,-94.279,69.366,176.6898,3.5102,-11710.8371
C00575=-23.215,-96.325,69.740,177.7754,0.8490,-11713.5503
C00576=-29.126,-95.625,70.117,179.8441,-0.0004,-11716.9400
C00577=-35.216,-93.589,70.366,179.9819,0.0007,-11720.6205
C00578=-41.276,-91.079,70.366,179.9820,0.0019,-11724.3795
C00579=-47.022,-88.212,70.117,179.8436,-0.0010,-11728.0601
C00580=-51.697,-84.528,69.740,177.7771,-0.8446,-11731.4498
C00581=-53.903,-79.427,69.366,176.6864,-3.5117,-11734.1627
C00582=-53.229,-73.964,68.906,178.2928,-7.4966,-11735.7411
C00583=-49.892,-68.885,68.033,179.7592,-7.6390,-11735.9150
C00584=-46.056,-63.647,66.266,179.8302,-6.2269,-11735.8901
C00585=-42.664,-58.966,63.969,179.7966,-4.0079,-11735.8871
C00586=-40.327,-55.279,61.754,-179.8773,0.9460,-11736.1114
C00587=-39.754,-52.385,60.163,-159.9107,19.0306,-11737.1942
C00588=-41.728,-49.608,59.535,-143.2689,5.7817,-11740.0690
C00589=-43.938,-47.576,59.508,-142.4189,-0.3039,-11742.7235
C00590=-45.791,-45.791,59.526,-142.4261,-0.0000,-11745.0000
C00591=-47.575,-43.938,59.508,-142.4189,0.3043,-11747.2759
C00592=-49.608,-41.728,59.535,-143.2694,-5.7917,-11749.9310
C00593=-52.385,-39.754,60.163,-159.9107,-19.0306,-11752.8058
C00594=-55.279,-40.327,61.754,-179.8773,-0.9460,-11753.8886
C00595=-58.966,-42.664,63.969,179.7966,4.0079,-11754.1129
C00596=-63.647,-46.056,66.266,179.8302,6.2269,-11754.1099
C00597=-68.885,-49.892,68.033,179.7592,7.6390,-11754.0850
C00598=-73.964,-53.229,68.906,178.2928,7.4966,-11754.2589
C00599=-79.427,-53.903,69.366,176.6864,3.5117,-11755.8373
C00600=-84.528,-51.697,69.740,177.7771,0.8446,-11758.5502
C00601=-88.212,-47.022,70.117,179.8436,0.0010,-11761.9399
C00602=-91.079,-41.276,70.366,179.9820,-0.0019,-11765.6205
C00603=-93.589,-35.216,70.366,179.9819,-0.0007,-11769.3795
C00604=-95.625,-29.126,70.117,179.8441,0.0004,-11773.0600
C00605=-96.325,-23.215,69.740,177.7754,-0.8490,-11776.4497
C00606=-94.279,-18.048,69.366,176.6898,-3.5102,-11779.1629
C00607=-89.940,-14.662,68.906,178.2885,-7.4940,-11780.7411
C00608=-83.988,-13.430,68.033,179.7593,-7.6388,-11780.9151
C00609=-77.571,-12.439,66.266,179.8289,-6.2253,-11780.8898
C00610=-71.864,-11.527,63.969,179.8008,-4.0103,-11780.8874
C00611=-67.603,-10.572,61.754,-179.8747,0.9417,-11781.1119
C00612=-65.152,-8.932,60.163,-159.9092,19.0297,-11782.1937
C00613=-64.584,-5.572,59.535,-143.2704,5.7854,-11785.0690
C00614=-64.710,-2.572,59.508,-142.4163,-0.3021,-11787.7239
C00615=-64.758,0.000,59.526,-142.4265,-0.0000,-11790.0000
C00616=-64.710,2.572,59.508,-142.4163,0.3021,-11792.2761
C00617=-64.584,5.572,59.535,-143.2704,-5.7854,-11794.9310
C00618=-65.152,8.932,60.163,-159.9092,-19.0297,-11797.8063
C00619=-67.603,10.572,61.754,-179.8747,-0.9417,-11798.8881
C00620=-71.864,11.527,63.969,179.8008,4.0103,-11799.1126
C00621=-77.571,12.439,66.266,179.8289,6.2253,-11799.1102
C00622=-83.988,13.430,68.033,179.7593,7.6388,-11799.0849
C00623=-89.940,14.662,68.906,178.2885,7.4940,-11799.2589
C00624=-94.279,18.048,69.366,176.6898,3.5102,-11800.8371
C00625=-96.325,23.215,69.740,177.7754,0.8490,-11803.5503
C00626=-95.625,29.126,70.117,179.8441,-0.0004,-11806.9400
C00627=-93.589,35.216,70.366,179.9819,0.0007,-11810.6205
C00628=-91.079,41.276,70.366,179.9820,0.0019,-11814.3795
C00629=-88.212,47.022,70.117,179.8436,-0.0010,-11818.0601
C00630=-84.528,51.697,69.740,177.7771,-0.8446,-11821.4498
C00631=-79.427,53.903,69.366,176.6864,-3.5117,-11824.1627
C00632=-73.964,53.229,68.906,178.2928,-7.4966,-11825.7411
C00633=-68.885,49.892,68.033,179.7592,-7.6390,-11825.9150
C00634=-63.647,46.056,66.266,179.8302,-6.2269,-11825.8901
C00635=-58.966,42.664,63.969,179.7966,-4.0079,-11825.8871
C00636=-55.279,40.327,61.754,-179.8773,0.9460,-11826.1114
C00637=-52.385,39.754,60.163,-159.9107,19.0306,-11827.1942
C00638=-49.608,41.728,59.535,-143.2689,5.7817,-11830.0690
C00639=-47.576,43.938,59.508,-142.4189,-0.3039,-11832.7235
C00640=-45.791,45.791,59.526,-142.4261,-0.0000,-11835.0000
C00641=-43.938,47.575,59.508,-142.4189,0.3043,-11837.2759
C00642=-41.728,49.608,59.535,-143.2694,-5.7917,-11839.9310
C00643=-39.754,52.385,60.163,-159.9107,-19.0306,-11842.8058
C00644=-40.327,55.279,61.754,-179.8773,-0.9460,-11843.8886
C00645=-42.664,58.966,63.969,179.7966,4.0079,-11844.1129
C00646=-46.056,63.647,66.266,179.8302,6.2269,-11844.1099
C00647=-49.892,68.885,68.033,179.7592,7.6390,-11844.0850
C00648=-53.229,73.964,68.906,178.2928,7.4966,-11844.2589
C00649=-53.903,79.427,69.366,176.6864,3.5117,-11845.8373
C00650=-51.697,84.528,69.740,177.7771,0.8446,-11848.5502
C00651=-47.022,88.212,70.117,179.8436,0.0010,-11851.9399
C00652=-41.276,91.079,70.366,179.9820,-0.0019,-11855.6205
C00653=-35.216,93.589,70.366,179.9819,-0.0007,-11859.3795
C00654=-29.126,95.625,70.117,179.8441,0.0004,-11863.0600
C00655=-23.215,96.325,69.740,177.7754,-0.8490,-11866.4497
C00656=-18.048,94.279,69.366,176.6898,-3.5102,-11869.1629
C00657=-14.662,89.940,68.906,178.2885,-7.4940,-11870.7411
C00658=-13.430,83.988,68.033,179.7593,-7.6388,-11870.9151
C00659=-12.439,77.571,66.266,179.8289,-6.2253,-11870.8898
C00660=-11.527,71.864,63.969,179.8008,-4.0103,-11870.8874
C00661=-10.572,67.603,61.754,-179.8747,0.9417,-11871.1119
C00662=-8.932,65.152,60.163,-159.9092,19.0297,-11872.1937
C00663=-5.572,64.584,59.535,-143.2704,5.7854,-11875.0690
C00664=-2.572,64.710,59.508,-142.4163,-0.3021,-11877.7239
C00665=0.000,64.758,59.526,-142.4265,0.0000,-11880.0000
C00666=0.000,63.425,61.276,-142.9995,0.0000,-11880.0000
C00667=2.450,63.381,61.257,-142.9908,0.3052,-11882.2137
C00668=5.367,63.268,61.285,-143.9210,-5.9690,-11884.8488
C00669=8.682,63.886,61.945,-161.3177,-18.5889,-11887.7390
C00670=10.270,66.465,63.612,-179.9745,-0.2474,-11888.7837
C00671=11.189,70.924,65.929,179.8229,4.1790,-11888.9651
C00672=12.084,76.878,68.324,179.8606,6.1406,-11888.9329
C00673=13.063,83.550,70.157,179.8074,7.4035,-11888.8862
C00674=14.270,89.726,71.060,178.4225,7.2562,-11889.0366
C00675=17.683,94.235,71.535,176.8235,3.4351,-11890.6278
C00676=22.929,96.378,71.920,177.8580,0.8281,-11893.3823
C00677=28.946,95.684,72.309,179.8513,0.0031,-11896.8314
C00678=35.156,93.612,72.565,179.9819,0.0007,-11900.5837
C00679=41.335,91.053,72.565,179.9820,0.0019,-11904.4165
C00680=47.191,88.127,72.309,179.8487,-0.0035,-11908.1685
C00681=51.936,84.362,71.920,177.8555,-0.8271,-11911.6178
C00682=54.130,79.138,71.535,176.8196,-3.4387,-11914.3719
C00683=53.356,73.536,71.060,178.4261,-7.2568,-11915.9638
C00684=49.842,68.316,70.157,179.8116,-7.4020,-11916.1137
C00685=45.816,62.906,68.324,179.8627,-6.1355,-11916.0668
C00686=42.239,58.063,65.929,179.8254,-4.1780,-11916.0347
C00687=39.736,54.260,63.612,-179.9731,0.2501,-11916.2163
C00688=39.035,51.313,61.945,-161.3213,18.5855,-11917.2611
C00689=40.942,48.532,61.285,-143.9220,5.9685,-11920.1513
C00690=43.085,46.550,61.257,-142.9899,-0.3005,-11922.7862
C00691=44.848,44.848,61.276,-143.0018,0.0000,-11925.0000
C00692=46.550,43.085,61.257,-142.9899,0.3005,-11927.2138
C00693=48.532,40.942,61.285,-143.9220,-5.9685,-11929.8487
C00694=51.313,39.035,61.945,-161.3213,-18.5855,-11932.7389
C00695=54.260,39.736,63.612,-179.9731,-0.2501,-11933.7837
C00696=58.063,42.239,65.929,179.8254,4.1780,-11933.9653
C00697=62.906,45.816,68.324,179.8627,6.1355,-11933.9332
C00698=68.316,49.842,70.157,179.8116,7.4020,-11933.8863
C00699=73.536,53.356,71.060,178.4261,7.2568,-11934.0362
C00700=79.138,54.130,71.535,176.8196,3.4387,-11935.6281
C00701=84.362,51.936,71.920,177.8555,0.8271,-11938.3822
C00702=88.127,47.191,72.309,179.8487,0.0035,-11941.8315
C00703=91.053,41.335,72.565,179.9820,-0.0019,-11945.5835
C00704=93.612,35.156,72.565,179.9819,-0.0007,-11949.4163
C00705=95.684,28.946,72.309,179.8513,-0.0031,-11953.1686
C00706=96.378,22.929,71.920,177.8580,-0.8281,-11956.6177
C00707=94.235,17.683,71.535,176.8235,-3.4351,-11959.3722
C00708=89.726,14.270,71.060,178.4225,-7.2562,-11960.9634
C00709=83.550,13.063,70.157,179.8074,-7.4035,-11961.1138
C00710=76.878,12.084,68.324,179.8606,-6.1406,-11961.0671
C00711=70.924,11.189,65.929,179.8229,-4.1790,-11961.0349
C00712=66.465,10.270,63.612,-179.9745,0.2474,-11961.2163
C00713=63.886,8.682,61.945,-161.3177,18.5889,-11962.2610
C00714=63.268,5.367,61.285,-143.9210,5.9690,-11965.1512
C00715=63.381,2.450,61.257,-142.9908,-0.3052,-11967.7863
C00716=63.425,0.000,61.276,-142.9995,0.0000,-11970.0000
C00717=63.381,-2.450,61.257,-142.9908,0.3052,-11972.2137
C00718=63.268,-5.367,61.285,-143.9210,-5.9690,-11974.8488
C00719=63.886,-8.682,61.945,-161.3234,-18.5881,-11977.7390
C00720=66.465,-10.270,63.612,-179.9745,-0.2474,-11978.7837
C00721=70.924,-11.189,65.929,179.8229,4.1790,-11978.9651
C00722=76.878,-12.084,68.324,179.8606,6.1406,-11978.9329
C00723=83.550,-13.063,70.157,179.8074,7.4035,-11978.8862
C00724=89.726,-14.270,71.060,178.4225,7.2562,-11979.0366
C00725=94.235,-17.683,71.535,176.8235,3.4351,-11980.6278
C00726=96.378,-22.929,71.920,177.8580,0.8281,-11983.3823
C00727=95.684,-28.946,72.309,179.8513,0.0031,-11986.8314
C00728=93.612,-35.156,72.565,179.9819,0.0007,-11990.5837
C00729=91.053,-41.335,72.565,179.9820,0.0019,-11994.4165
C00730=88.127,-47.191,72.309,179.8487,-0.0035,-11998.1685
C00731=84.362,-51.936,71.920,177.8555,-0.8271,-12001.6178
C00732=79.138,-54.130,71.535,176.8196,-3.4387,-12004.3719
C00733=73.536,-53.356,71.060,178.4261,-7.2568,-12005.9638
C00734=68.316,-49.842,70.157,179.8116,-7.4020,-12006.1137
C00735=62.906,-45.816,68.324,179.8627,-6.1355,-12006.0668
C00736=58.063,-42.239,65.929,179.8254,-4.1780,-12006.0347
C00737=54.260,-39.736,63.612,-179.9731,0.2501,-12006.2163
C00738=51.313,-39.035,61.945,-161.3213,18.5855,-12007.2611
C00739=48.532,-40.942,61.285,-143.9220,5.9685,-12010.1513
C00740=46.550,-43.085,61.257,-142.9899,-0.3005,-12012.7862
C00741=44.848,-44.848,61.276,-143.0018,0.0000,-12015.0000
C00742=43.085,-46.550,61.257,-142.9899,0.3005,-12017.2138
C00743=40.942,-48.532,61.285,-143.9220,-5.9685,-12019.8487
C00744=39.035,-51.313,61.945,-161.3213,-18.5855,-12022.7389
C00745=39.736,-54.260,63.612,-179.9731,-0.2501,-12023.7837
C00746=42.239,-58.063,65.929,179.8254,4.1780,-12023.9653
C00747=45.816,-62.906,68.324,179.8627,6.1355,-12023.9332
C00748=49.842,-68.316,70.157,179.8116,7.4020,-12023.8863
C00749=53.356,-73.536,71.060,178.4261,7.2568,-12024.0362
C00750=54.130,-79.138,71.535,176.8196,3.4387,-12025.6281
C00751=51.936,-84.362,71.920,177.8555,0.8271,-12028.3822
C00752=47.191,-88.127,72.309,179.8487,0.0035,-12031.8315
C00753=41.335,-91.053,72.565,179.9820,-0.0019,-12035.5835
C00754=35.156,-93.612,72.565,179.9819,-0.0007,-12039.4163
C00755=28.946,-95.684,72.309,179.8513,-0.0031,-12043.1686
C00756=22.929,-96.378,71.920,177.8580,-0.8281,-12046.6177
C00757=17.683,-94.235,71.535,176.8235,-3.4351,-12049.3722
C00758=14.270,-89.726,71.060,178.4225,-7.2562,-12050.9634
C00759=13.063,-83.550,70.157,179.8074,-7.4035,-12051.1138
C00760=12.084,-76.878,68.324,179.8606,-6.1406,-12051.0671
C00761=11.189,-70.924,65.929,179.8229,-4.1790,-12051.0349
C00762=10.270,-66.465,63.612,-179.9745,0.2474,-12051.2163
C00763=8.682,-63.886,61.945,-161.3177,18.5889,-12052.2610
C00764=5.367,-63.268,61.285,-143.9210,5.9690,-12055.1512
C00765=2.450,-63.381,61.257,-142.9908,-0.3052,-12057.7863
C00766=0.000,-63.425,61.276,-142.9995,0.0000,-12060.0000
C00767=0.000,-63.425,61.276,-142.9995,0.0000,-12060.0000
C00768=-2.450,-63.381,61.257,-142.9908,0.3052,-12062.2137
C00769=-5.367,-63.268,61.285,-143.9210,-5.9690,-12064.8488
C00770=-8.682,-63.886,61.945,-161.3234,-18.5881,-12067.7390
C00771=-10.270,-66.465,63.612,-179.9745,-0.2474,-12068.7837
C00772=-11.189,-70.924,65.929,179.8229,4.1790,-12068.9651
C00773=-12.084,-76.878,68.324,179.8606,6.1406,-12068.9329
C00774=-13.063,-83.550,70.157,179.8074,7.4035,-12068.8862
C00775=-14.270,-89.726,71.060,178.4225,7.2562,-12069.0366
C00776=-17.683,-94.235,71.535,176.8235,3.4351,-12070.6278
C00777=-22.929,-96.378,71.920,177.8580,0.8281,-12073.3823
C00778=-28.946,-95.684,72.309,179.8513,0.0031,-12076.8314
C00779=-35.156,-93.612,72.565,179.9819,0.0007,-12080.5837
C00780=-41.335,-91.053,72.565,179.9820,0.0019,-12084.4165
C00781=-47.191,-88.127,72.309,179.8487,-0.0035,-12088.1685
C00782=-51.936,-84.362,71.920,177.8555,-0.8271,-12091.6178
C00783=-54.130,-79.138,71.535,176.8196,-3.4387,-12094.3719
C00784=-53.356,-73.536,71.060,178.4261,-7.2568,-12095.9638
C00785=-49.842,-68.316,70.157,179.8116,-7.4020,-12096.1137
C00786=-45.816,-62.906,68.324,179.8627,-6.1355,-12096.0668
C00787=-42.239,-58.063,65.929,179.8254,-4.1780,-12096.0347
C00788=-39.736,-54.260,63.612,-179.9731,0.2501,-12096.2163
C00789=-39.035,-51.313,61.945,-161.3213,18.5855,-12097.2611
C00790=-40.942,-48.532,61.285,-143.9220,5.9685,-12100.1513
C00791=-43.085,-46.550,61.257,-142.9899,-0.3005,-12102.7862
C00792=-44.848,-44.848,61.276,-143.0018,0.0000,-12105.0000
C00793=-46.550,-43.085,61.257,-142.9899,0.3005,-12107.2138
C00794=-48.532,-40.942,61.285,-143.9220,-5.9685,-12109.8487
C00795=-51.313,-39.035,61.945,-161.3213,-18.5855,-12112.7389
C00796=-54.260,-39.736,63.612,-179.9731,-0.2501,-12113.7837
C00797=-58.063,-42.239,65.929,179.8254,4.1780,-12113.9653
C00798=-62.906,-45.816,68.324,179.8627,6.1355,-12113.9332
C00799=-68.316,-49.842,70.157,179.8116,7.4020,-12113.8863
C00800=-73.536,-53.356,71.060,178.4261,7.2568,-12114.0362
C00801=-79.138,-54.130,71.535,176.8196,3.4387,-12115.6281
C00802=-84.362,-51.936,71.920,177.8555,0.8271,-12118.3822
C00803=-88.127,-47.191,72.309,179.8487,0.0035,-12121.8315
C00804=-91.053,-41.335,72.565,179.9820,-0.0019,-12125.5835
C00805=-93.612,-35.156,72.565,179.9819,-0.0007,-12129.4163
C00806=-95.684,-28.946,72.309,179.8513,-0.0031,-12133.1686
C00807=-96.378,-22.929,71.920,177.8580,-0.8281,-12136.6177
C00808=-94.235,-17.683,71.535,176.8235,-3.4351,-12139.3722
C00809=-89.726,-14.270,71.060,178.4225,-7.2562,-12140.9634
C00810=-83.550,-13.063,70.157,179.8074,-7.4035,-12141.1138
C00811=-76.878,-12.084,68.324,179.8606,-6.1406,-12141.0671
C00812=-70.924,-11.189,65.929,179.8229,-4.1790,-12141.0349
C00813=-66.465,-10.270,63.612,-179.9745,0.2474,-12141.2163
C00814=-63.886,-8.682,61.945,-161.3177,18.5889,-12142.2610
C00815=-63.268,-5.367,61.285,-143.9210,5.9690,-12145.1512
C00816=-63.381,-2.450,61.257,-142.9908,-0.3052,-12147.7863
C00817=-63.425,0.000,61.276,-142.9995,0.0000,-12150.0000
C00818=-63.381,2.450,61.257,-142.9908,0.3052,-12152.2137
C00819=-63.268,5.367,61.285,-143.9210,-5.9690,-12154.8488
C00820=-63.886,8.682,61.945,-161.3234,-18.5881,-12157.7390
C00821=-66.465,10.270,63.612,-179.9745,-0.2474,-12158.7837
C00822=-70.924,11.189,65.929,179.8229,4.1790,-12158.9651
C00823=-76.878,12.084,68.324,179.8606,6.1406,-12158.9329
C00824=-83.550,13.063,70.157,179.8074,7.4035,-12158.8862
C00825=-89.726,14.270,71.060,178.4225,7.2562,-12159.0366
C00826=-94.235,17.683,71.535,176.8235,3.4351,-12160.6278
C00827=-96.378,22.929,71.920,177.8580,0.8281,-12163.3823
C00828=-95.684,28.946,72.309,179.8513,0.0031,-12166.8314
C00829=-93.612,35.156,72.565,179.9819,0.0007,-12170.5837
C00830=-91.053,41.335,72.565,179.9820,0.0019,-12174.4165
C00831=-88.127,47.191,72.309,179.8487,-0.0035,-12178.1685
C00832=-84.362,51.936,71.920,177.8555,-0.8271,-12181.6178
C00833=-79.138,54.130,71.535,176.8196,-3.4387,-12184.3719
C00834=-73.536,53.356,71.060,178.4261,-7.2568,-12185.9638
C00835=-68.316,49.842,70.157,179.8116,-7.4020,-12186.1137
C00836=-62.906,45.816,68.324,179.8627,-6.1355,-12186.0668
C00837=-58.063,42.239,65.929,179.8254,-4.1780,-12186.0347
C00838=-54.260,39.736,63.612,-179.9731,0.2501,-12186.2163
C00839=-51.313,39.035,61.945,-161.3213,18.5855,-12187.2611
C00840=-48.532,40.942,61.285,-143.9220,5.9685,-12190.1513
C00841=-46.550,43.085,61.257,-142.9899,-0.3005,-12192.7862
C00842=-44.848,44.848,61.276,-143.0018,-0.0000,-12195.0000
C00843=-43.085,46.550,61.257,-142.9899,0.3005,-12197.2138
C00844=-40.942,48.532,61.285,-143.9220,-5.9685,-12199.8487
C00845=-39.035,51.313,61.945,-161.3213,-18.5855,-12202.7389
C00846=-39.736,54.260,63.612,-179.9731,-0.2501,-12203.7837
C00847=-42.239,58.063,65.929,179.8254,4.1780,-12203.9653
C00848=-45.816,62.906,68.324,179.8627,6.1355,-12203.9332
C00849=-49.842,68.316,70.157,179.8116,7.4020,-12203.8863
C00850=-53.356,73.536,71.060,178.4261,7.2568,-12204.0362
C00851=-54.130,79.138,71.535,176.8196,3.4387,-12205.6281
C00852=-51.936,84.362,71.920,177.8555,0.8271,-12208.3822
C00853=-47.191,88.127,72.309,179.8487,0.0035,-12211.8315
C00854=-41.335,91.053,72.565,179.9820,-0.0019,-12215.5835
C00855=-35.156,93.612,72.565,179.9819,-0.0007,-12219.4163
C00856=-28.946,95.684,72.309,179.8513,-0.0031,-12223.1686
C00857=-22.929,96.378,71.920,177.8580,-0.8281,-12226.6177
C00858=-17.683,94.235,71.535,176.8235,-3.4351,-12229.3722
C00859=-14.270,89.726,71.060,178.4225,-7.2562,-12230.9634
C00860=-13.063,83.550,70.157,179.8074,-7.4035,-12231.1138
C00861=-12.084,76.878,68.324,179.8606,-6.1406,-12231.0671
C00862=-11.189,70.924,65.929,179.8229,-4.1790,-12231.0349
C00863=-10.270,66.465,63.612,-179.9745,0.2474,-12231.2163
C00864=-8.682,63.886,61.945,-161.3234,18.5881,-12232.2610
C00865=-5.367,63.268,61.285,-143.9210,5.9690,-12235.1512
C00866=-2.450,63.381,61.257,-142.9908,-0.3052,-12237.7863
C00867=0.000,63.425,61.276,-142.9995,-0.0000,-12240.0000
C00868=0.000,62.111,63.041,-143.6744,-0.0000,-12240.0000
C00869=2.330,62.072,63.021,-143.6676,0.2972,-12242.1497
C00870=5.165,61.970,63.050,-144.6738,-6.1198,-12244.7644
C00871=8.436,62.639,63.741,-162.7278,-18.0361,-12247.6702
C00872=9.975,65.350,65.485,179.9678,0.3585,-12248.6786
C00873=10.861,70.011,67.904,179.8507,4.2771,-12248.8182
C00874=11.743,76.212,70.393,179.8893,5.9934,-12248.7594
C00875=12.712,83.133,72.289,179.8539,7.1060,-12248.6938
C00876=13.898,89.524,73.219,178.5603,6.9499,-12248.8243
C00877=17.338,94.193,73.707,176.9802,3.3227,-12250.4296
C00878=22.659,96.427,74.103,177.9563,0.7984,-12253.2238
C00879=28.778,95.739,74.502,179.8568,0.0012,-12256.7302
C00880=35.099,93.634,74.765,179.9819,0.0007,-12260.5487
C00881=41.391,91.028,74.765,179.9820,0.0019,-12264.4516
C00882=47.349,88.047,74.502,179.8564,-0.0009,-12268.2700
C00883=52.162,84.206,74.103,177.9559,-0.7970,-12271.7764
C00884=54.344,78.865,73.707,176.9785,-3.3216,-12274.5698
C00885=53.475,73.130,73.219,178.5593,-6.9449,-12276.1755
C00886=49.795,67.773,72.289,179.8532,-7.1065,-12276.3059
C00887=45.586,62.194,70.393,179.8921,-5.9921,-12276.2401
C00888=41.825,57.185,67.904,179.8469,-4.2793,-12276.1817
C00889=39.156,53.262,65.485,179.9645,-0.3579,-12276.3218
C00890=38.328,50.258,63.741,-162.7241,18.0404,-12277.3300
C00891=40.167,47.472,63.050,-144.6731,6.1175,-12280.2352
C00892=42.244,45.539,63.021,-143.6668,-0.2954,-12282.8504
C00893=43.919,43.919,63.041,-143.6737,-0.0000,-12285.0000
C00894=45.539,42.244,63.021,-143.6668,0.2954,-12287.1496
C00895=47.472,40.167,63.050,-144.6767,-6.1220,-12289.7648
C00896=50.258,38.328,63.741,-162.7241,-18.0404,-12292.6700
C00897=53.262,39.156,65.485,179.9645,0.3579,-12293.6782
C00898=57.185,41.825,67.904,179.8469,4.2793,-12293.8183
C00899=62.194,45.586,70.393,179.8921,5.9921,-12293.7599
C00900=67.773,49.795,72.289,179.8532,7.1065,-12293.6941
C00901=73.130,53.475,73.219,178.5593,6.9449,-12293.8245
C00902=78.865,54.344,73.707,176.9785,3.3216,-12295.4302
C00903=84.206,52.162,74.103,177.9559,0.7970,-12298.2236
C00904=88.047,47.349,74.502,179.8564,0.0009,-12301.7300
C00905=91.028,41.391,74.765,179.9820,-0.0019,-12305.5484
C00906=93.634,35.099,74.765,179.9819,-0.0007,-12309.4513
C00907=95.739,28.778,74.502,179.8568,-0.0012,-12313.2698
C00908=96.427,22.659,74.103,177.9563,-0.7984,-12316.7762
C00909=94.193,17.338,73.707,176.9802,-3.3227,-12319.5704
C00910=89.524,13.898,73.219,178.5603,-6.9499,-12321.1757
C00911=83.133,12.712,72.289,179.8539,-7.1060,-12321.3062
C00912=76.212,11.743,70.393,179.8893,-5.9934,-12321.2406
C00913=70.011,10.861,67.904,179.8507,-4.2771,-12321.1818
C00914=65.350,9.975,65.485,179.9678,-0.3585,-12321.3214
C00915=62.639,8.436,63.741,-162.7278,18.0361,-12322.3298
C00916=61.970,5.165,63.050,-144.6738,6.1198,-12325.2356
C00917=62.072,2.330,63.021,-143.6676,-0.2972,-12327.8503
C00918=62.111,0.000,63.041,-143.6744,-0.0000,-12330.0000
C00919=62.072,-2.330,63.021,-143.6676,0.2972,-12332.1497
C00920=61.970,-5.165,63.050,-144.6738,-6.1198,-12334.7644
C00921=62.640,-8.436,63.741,-162.7277,-18.0361,-12337.6701
C00922=65.350,-9.975,65.485,179.9678,0.3585,-12338.6786
C00923=70.011,-10.861,67.904,179.8507,4.2771,-12338.8182
C00924=76.212,-11.743,70.393,179.8893,5.9934,-12338.7594
C00925=83.133,-12.712,72.289,179.8539,7.1060,-12338.6938
C00926=89.524,-13.898,73.219,178.5603,6.9499,-12338.8243
C00927=94.193,-17.338,73.707,176.9802,3.3227,-12340.4296
C00928=96.427,-22.659,74.103,177.9563,0.7984,-12343.2238
C00929=95.739,-28.778,74.502,179.8568,0.0012,-12346.7302
C00930=93.634,-35.099,74.765,179.9819,0.0007,-12350.5487
C00931=91.028,-41.391,74.765,179.9820,0.0019,-12354.4516
C00932=88.047,-47.349,74.502,179.8564,-0.0009,-12358.2700
C00933=84.206,-52.162,74.103,177.9559,-0.7970,-12361.7764
C00934=78.865,-54.344,73.707,176.9785,-3.3216,-12364.5698
C00935=73.130,-53.475,73.219,178.5593,-6.9449,-12366.1755
C00936=67.773,-49.795,72.289,179.8532,-7.1065,-12366.3059
C00937=62.194,-45.586,70.393,179.8921,-5.9921,-12366.2401
C00938=57.185,-41.825,67.904,179.8469,-4.2793,-12366.1817
C00939=53.262,-39.156,65.485,179.9645,-0.3579,-12366.3218
C00940=50.258,-38.328,63.741,-162.7241,18.0404,-12367.3300
C00941=47.472,-40.167,63.050,-144.6731,6.1175,-12370.2352
C00942=45.539,-42.244,63.021,-143.6668,-0.2954,-12372.8504
C00943=43.919,-43.919,63.041,-143.6737,0.0000,-12375.0000
C00944=42.244,-45.539,63.021,-143.6668,0.2954,-12377.1496
C00945=40.167,-47.472,63.050,-144.6767,-6.1220,-12379.7648
C00946=38.328,-50.258,63.741,-162.7241,-18.0404,-12382.6700
C00947=39.156,-53.262,65.485,179.9645,0.3579,-12383.6782
C00948=41.825,-57.185,67.904,179.8469,4.2793,-12383.8183
C00949=45.586,-62.194,70.393,179.8921,5.9921,-12383.7599
C00950=49.795,-67.773,72.289,179.8532,7.1065,-12383.6941
C00951=53.475,-73.130,73.219,178.5593,6.9449,-12383.8245
C00952=54.344,-78.865,73.707,176.9785,3.3216,-12385.4302
C00953=52.162,-84.206,74.103,177.9559,0.7970,-12388.2236
C00954=47.349,-88.047,74.502,179.8564,0.0009,-12391.7300
C00955=41.391,-91.028,74.765,179.9820,-0.0019,-12395.5484
C00956=35.099,-93.634,74.765,179.9819,-0.0007,-12399.4513
C00957=28.778,-95.739,74.502,179.8568,-0.0012,-12403.2698
C00958=22.659,-96.427,74.103,177.9563,-0.7984,-12406.7762
C00959=17.338,-94.193,73.707,176.9802,-3.3227,-12409.5704
C00960=13.898,-89.524,73.219,178.5603,-6.9499,-12411.1757
C00961=12.712,-83.133,72.289,179.8539,-7.1060,-12411.3062
C00962=11.743,-76.212,70.393,179.8893,-5.9934,-12411.2406
C00963=10.861,-70.011,67.904,179.8507,-4.2771,-12411.1818
C00964=9.975,-65.350,65.485,179.9678,-0.3585,-12411.3214
C00965=8.436,-62.639,63.741,-162.7278,18.0361,-12412.3298
C00966=5.165,-61.970,63.050,-144.6738,6.1198,-12415.2356
C00967=2.330,-62.072,63.021,-143.6676,-0.2972,-12417.8503
C00968=0.000,-62.111,63.041,-143.6744,0.0000,-12420.0000
C00969=0.000,-62.111,63.041,-143.6744,0.0000,-12420.0000
C00970=-2.330,-62.072,63.021,-143.6676,0.2972,-12422.1497
C00971=-5.165,-61.970,63.050,-144.6738,-6.1198,-12424.7644
C00972=-8.436,-62.640,63.741,-162.7277,-18.0361,-12427.6701
C00973=-9.975,-65.350,65.485,179.9678,0.3585,-12428.6786
C00974=-10.861,-70.011,67.904,179.8507,4.2771,-12428.8182
C00975=-11.743,-76.212,70.393,179.8893,5.9934,-12428.7594
C00976=-12.712,-83.133,72.289,179.8539,7.1060,-12428.6938
C00977=-13.898,-89.524,73.219,178.5603,6.9499,-12428.8243
C00978=-17.338,-94.193,73.707,176.9802,3.3227,-12430.4296
C00979=-22.659,-96.427,74.103,177.9563,0.7984,-12433.2238
C00980=-28.778,-95.739,74.502,179.8568,0.0012,-12436.7302
C00981=-35.099,-93.634,74.765,179.9819,0.0007,-12440.5487
C00982=-41.391,-91.028,74.765,179.9820,0.0019,-12444.4516
C00983=-47.349,-88.047,74.502,179.8564,-0.0009,-12448.2700
C00984=-52.162,-84.206,74.103,177.9559,-0.7970,-12451.7764
C00985=-54.344,-78.865,73.707,176.9785,-3.3216,-12454.5698
C00986=-53.475,-73.130,73.219,178.5593,-6.9449,-12456.1755
C00987=-49.795,-67.773,72.289,179.8532,-7.1065,-12456.3059
C00988=-45.586,-62.194,70.393,179.8921,-5.9921,-12456.2401
C00989=-41.825,-57.185,67.904,179.8469,-4.2793,-12456.1817
C00990=-39.156,-53.262,65.485,179.9645,-0.3579,-12456.3218
C00991=-38.328,-50.258,63.741,-162.7241,18.0404,-12457.3300
C00992=-40.167,-47.472,63.050,-144.6731,6.1175,-12460.2352
C00993=-42.244,-45.539,63.021,-143.6668,-0.2954,-12462.8504
C00994=-43.919,-43.919,63.041,-143.6737,0.0000,-12465.0000
C00995=-45.539,-42.244,63.021,-143.6668,0.2954,-12467.1496
C00996=-47.472,-40.167,63.050,-144.6767,-6.1220,-12469.7648
C00997=-50.258,-38.328,63.741,-162.7241,-18.0404,-12472.6700
C00998=-53.262,-39.156,65.485,179.9645,0.3579,-12473.6782
C00999=-57.185,-41.825,67.904,179.8469,4.2793,-12473.8183
C01000=-62.194,-45.586,70.393,179.8921,5.9921,-12473.7599
C01001=-67.773,-49.795,72.289,179.8532,7.1065,-12473.6941
C01002=-73.130,-53.475,73.219,178.5593,6.9449,-12473.8245
C01003=-78.865,-54.344,73.707,176.9785,3.3216,-12475.4302
C01004=-84.206,-52.162,74.103,177.9559,0.7970,-12478.2236
C01005=-88.047,-47.349,74.502,179.8564,0.0009,-12481.7300
C01006=-91.028,-41.391,74.765,179.9820,-0.0019,-12485.5484
C01007=-93.634,-35.099,74.765,179.9819,-0.0007,-12489.4513
C01008=-95.739,-28.778,74.502,179.8568,-0.0012,-12493.2698
C01009=-96.427,-22.659,74.103,177.9563,-0.7984,-12496.7762
C01010=-94.193,-17.338,73.707,176.9802,-3.3227,-12499.5704
C01011=-89.524,-13.898,73.219,178.5603,-6.9499,-12501.1757
C01012=-83.133,-12.712,72.289,179.8539,-7.1060,-12501.3062
C01013=-76.212,-11.743,70.393,179.8893,-5.9934,-12501.2406
C01014=-70.011,-10.861,67.904,179.8507,-4.2771,-12501.1818
C01015=-65.350,-9.975,65.485,179.9678,-0.3585,-12501.3214
C01016=-62.639,-8.436,63.741,-162.7278,18.0361,-12502.3298
C01017=-61.970,-5.165,63.050,-144.6738,6.1198,-12505.2356
C01018=-62.072,-2.330,63.021,-143.6676,-0.2972,-12507.8503
C01019=-62.111,0.000,63.041,-143.6744,0.0000,-12510.0000
C01020=-62.072,2.330,63.021,-143.6676,0.2972,-12512.1497
C01021=-61.970,5.165,63.050,-144.6738,-6.1198,-12514.7644
C01022=-62.640,8.436,63.741,-162.7277,-18.0361,-12517.6701
C01023=-65.350,9.975,65.485,179.9678,0.3585,-12518.6786
C01024=-70.011,10.861,67.904,179.8507,4.2771,-12518.8182
C01025=-76.212,11.743,70.393,179.8893,5.9934,-12518.7594
C01026=-83.133,12.712,72.289,179.8539,7.1060,-12518.6938
C01027=-89.524,13.898,73.219,178.5603,6.9499,-12518.8243
C01028=-94.193,17.338,73.707,176.9802,3.3227,-12520.4296
C01029=-96.427,22.659,74.103,177.9563,0.7984,-12523.2238
C01030=-95.739,28.778,74.502,179.8568,0.0012,-12526.7302
C01031=-93.634,35.099,74.765,179.9819,0.0007,-12530.5487
C01032=-91.028,41.391,74.765,179.9820,0.0019,-12534.4516
C01033=-88.047,47.349,74.502,179.8564,-0.0009,-12538.2700
C01034=-84.206,52.162,74.103,177.9559,-0.7970,-12541.7764
C01035=-78.865,54.344,73.707,176.9785,-3.3216,-12544.5698
C01036=-73.130,53.475,73.219,178.5593,-6.9449,-12546.1755
C01037=-67.773,49.795,72.289,179.8532,-7.1065,-12546.3059
C01038=-62.194,45.586,70.393,179.8921,-5.9921,-12546.2401
C01039=-57.185,41.825,67.904,179.8469,-4.2793,-12546.1817
C01040=-53.262,39.156,65.485,179.9645,-0.3579,-12546.3218
C01041=-50.258,38.328,63.741,-162.7241,18.0404,-12547.3300
C01042=-47.472,40.167,63.050,-144.6731,6.1175,-12550.2352
C01043=-45.539,42.244,63.021,-143.6668,-0.2954,-12552.8504
C01044=-43.919,43.919,63.041,-143.6737,0.0000,-12555.0000
C01045=-42.244,45.539,63.021,-143.6668,0.2954,-12557.1496
C01046=-40.167,47.472,63.050,-144.6767,-6.1220,-12559.7648
C01047=-38.328,50.258,63.741,-162.7241,-18.0404,-12562.6700
C01048=-39.156,53.262,65.485,179.9645,0.3579,-12563.6782
C01049=-41.825,57.185,67.904,179.8469,4.2793,-12563.8183
C01050=-45.586,62.194,70.393,179.8921,5.9921,-12563.7599
C01051=-49.795,67.773,72.289,179.8532,7.1065,-12563.6941
C01052=-53.475,73.130,73.219,178.5593,6.9449,-12563.8245
C01053=-54.344,78.865,73.707,176.9785,3.3216,-12565.4302
C01054=-52.162,84.206,74.103,177.9559,0.7970,-12568.2236
C01055=-47.349,88.047,74.502,179.8564,0.0009,-12571.7300
C01056=-41.391,91.028,74.765,179.9820,-0.0019,-12575.5484
C01057=-35.099,93.634,74.765,179.9819,-0.0007,-12579.4513
C01058=-28.778,95.739,74.502,179.8568,-0.0012,-12583.2698
C01059=-22.659,96.427,74.103,177.9563,-0.7984,-12586.7762
C01060=-17.338,94.193,73.707,176.9802,-3.3227,-12589.5704
C01061=-13.898,89.524,73.219,178.5603,-6.9499,-12591.1757
C01062=-12.712,83.133,72.289,179.8539,-7.1060,-12591.3062
C01063=-11.743,76.212,70.393,179.8893,-5.9934,-12591.2406
C01064=-10.861,70.011,67.904,179.8507,-4.2771,-12591.1818
C01065=-9.975,65.350,65.485,179.9678,-0.3585,-12591.3214
C01066=-8.436,62.640,63.741,-162.7277,18.0361,-12592.3299
C01067=-5.165,61.970,63.050,-144.6738,6.1198,-12595.2356
C01068=-2.330,62.072,63.021,-143.6676,-0.2972,-12597.8503
C01069=0.000,62.111,63.041,-143.6744,0.0000,-12600.0000
C01070=0.000,60.820,64.822,-144.4503,0.0000,-12600.0000
C01071=2.212,60.785,64.801,-144.4407,0.2926,-12602.0841
C01072=4.967,60.695,64.832,-145.5318,-6.2395,-12604.6784
C01073=8.195,61.417,65.554,-164.1096,-17.3895,-12607.6002
C01074=9.686,64.262,67.375,179.9289,0.8741,-12608.5715
C01075=10.544,69.129,69.894,179.8743,4.3120,-12608.6723
C01076=11.418,75.576,72.474,179.9164,5.7880,-12608.5913
C01077=12.382,82.740,74.428,179.8876,6.7409,-12608.5111
C01078=13.550,89.334,75.383,178.6906,6.5704,-12608.6248
C01079=17.016,94.154,75.883,177.1656,3.1658,-12610.2442
C01080=22.407,96.473,76.288,178.0701,0.7603,-12613.0758
C01081=28.621,95.791,76.696,179.8623,-0.0007,-12616.6354
C01082=35.046,93.654,76.964,179.9819,0.0007,-12620.5162
C01083=41.442,91.005,76.964,179.9820,0.0019,-12624.4836
C01084=47.497,87.973,76.696,179.8642,0.0017,-12628.3648
C01085=52.372,84.060,76.288,178.0752,-0.7593,-12631.9242
C01086=54.545,78.609,75.883,177.1688,-3.1633,-12634.7559
C01087=53.588,72.750,75.383,178.6911,-6.5728,-12636.3755
C01088=49.751,67.261,74.428,179.8915,-6.7417,-12636.4893
C01089=45.367,61.514,72.474,179.9177,-5.7873,-12636.4090
C01090=41.426,56.337,69.894,179.8743,-4.3140,-12636.3280
C01091=38.591,52.289,67.375,179.9265,-0.8715,-12636.4285
C01092=37.634,49.223,65.554,-164.1107,17.3872,-12637.4001
C01093=39.406,46.429,64.832,-145.5293,6.2383,-12640.3225
C01094=41.417,44.545,64.801,-144.4394,-0.2887,-12642.9160
C01095=43.006,43.006,64.822,-144.4511,-0.0000,-12645.0000
C01096=44.545,41.417,64.801,-144.4394,0.2887,-12647.0840
C01097=46.430,39.405,64.832,-145.5330,-6.2436,-12649.6788
C01098=49.223,37.634,65.554,-164.1107,-17.3872,-12652.5999
C01099=52.289,38.591,67.375,179.9265,0.8715,-12653.5715
C01100=56.337,41.426,69.894,179.8743,4.3140,-12653.6720
C01101=61.514,45.367,72.474,179.9177,5.7873,-12653.5910
C01102=67.261,49.751,74.428,179.8915,6.7417,-12653.5107
C01103=72.750,53.588,75.383,178.6911,6.5728,-12653.6245
C01104=78.609,54.545,75.883,177.1688,3.1633,-12655.2441
C01105=84.060,52.372,76.288,178.0752,0.7593,-12658.0758
C01106=87.973,47.497,76.696,179.8642,-0.0017,-12661.6352
C01107=91.005,41.442,76.964,179.9820,-0.0019,-12665.5164
C01108=93.654,35.046,76.964,179.9819,-0.0007,-12669.4838
C01109=95.791,28.621,76.696,179.8623,0.0007,-12673.3646
C01110=96.473,22.407,76.288,178.0701,-0.7603,-12676.9242
C01111=94.154,17.016,75.883,177.1656,-3.1658,-12679.7558
C01112=89.334,13.550,75.383,178.6906,-6.5704,-12681.3752
C01113=82.740,12.382,74.428,179.8876,-6.7409,-12681.4889
C01114=75.576,11.418,72.474,179.9164,-5.7880,-12681.4087
C01115=69.129,10.544,69.894,179.8743,-4.3120,-12681.3277
C01116=64.262,9.686,67.375,179.9289,-0.8741,-12681.4285
C01117=61.417,8.195,65.554,-164.1096,17.3895,-12682.3998
C01118=60.695,4.967,64.832,-145.5318,6.2395,-12685.3216
C01119=60.785,2.212,64.801,-144.4407,-0.2926,-12687.9159
C01120=60.820,0.000,64.822,-144.4503,-0.0000,-12690.0000
C01121=60.785,-2.212,64.801,-144.4407,0.2926,-12692.0841
C01122=60.695,-4.967,64.832,-145.5318,-6.2395,-12694.6784
C01123=61.417,-8.195,65.554,-164.1096,-17.3895,-12697.6002
C01124=64.262,-9.686,67.375,179.9289,0.8741,-12698.5715
C01125=69.129,-10.544,69.894,179.8743,4.3120,-12698.6723
C01126=75.576,-11.418,72.474,179.9164,5.7880,-12698.5913
C01127=82.740,-12.382,74.428,179.8876,6.7409,-12698.5111
C01128=89.334,-13.550,75.383,178.6906,6.5704,-12698.6248
C01129=94.154,-17.016,75.883,177.1656,3.1658,-12700.2442
C01130=96.473,-22.407,76.288,178.0701,0.7603,-12703.0758
C01131=95.791,-28.621,76.696,179.8623,-0.0007,-12706.6354
C01132=93.654,-35.046,76.964,179.9819,0.0007,-12710.5162
C01133=91.005,-41.442,76.964,179.9820,0.0019,-12714.4836
C01134=87.973,-47.497,76.696,179.8642,0.0017,-12718.3648
C01135=84.060,-52.372,76.288,178.0752,-0.7593,-12721.9242
C01136=78.609,-54.545,75.883,177.1688,-3.1633,-12724.7559
C01137=72.750,-53.588,75.383,178.6911,-6.5728,-12726.3755
C01138=67.261,-49.751,74.428,179.8915,-6.7417,-12726.4893
C01139=61.514,-45.367,72.474,179.9177,-5.7873,-12726.4090
C01140=56.337,-41.426,69.894,179.8743,-4.3140,-12726.3280
C01141=52.289,-38.591,67.375,179.9265,-0.8715,-12726.4285
C01142=49.223,-37.634,65.554,-164.1107,17.3872,-12727.4001
C01143=46.429,-39.406,64.832,-145.5293,6.2383,-12730.3225
C01144=44.545,-41.417,64.801,-144.4394,-0.2887,-12732.9160
C01145=43.006,-43.006,64.822,-144.4511,-0.0000,-12735.0000
C01146=41.417,-44.545,64.801,-144.4394,0.2887,-12737.0840
C01147=39.405,-46.430,64.832,-145.5330,-6.2436,-12739.6788
C01148=37.634,-49.223,65.554,-164.1107,-17.3872,-12742.5999
C01149=38.591,-52.289,67.375,179.9265,0.8715,-12743.5715
C01150=41.426,-56.337,69.894,179.8743,4.3140,-12743.6720
C01151=45.367,-61.514,72.474,179.9177,5.7873,-12743.5910
C01152=49.751,-67.261,74.428,179.8915,6.7417,-12743.5107
C01153=53.588,-72.750,75.383,178.6911,6.5728,-12743.6245
C01154=54.545,-78.609,75.883,177.1688,3.1633,-12745.2441
C01155=52.372,-84.060,76.288,178.0752,0.7593,-12748.0758
C01156=47.497,-87.973,76.696,179.8642,-0.0017,-12751.6352
C01157=41.442,-91.005,76.964,179.9820,-0.0019,-12755.5164
C01158=35.046,-93.654,76.964,179.9819,-0.0007,-12759.4838
C01159=28.621,-95.791,76.696,179.8623,0.0007,-12763.3646
C01160=22.407,-96.473,76.288,178.0701,-0.7603,-12766.9242
C01161=17.016,-94.154,75.883,177.1656,-3.1658,-12769.7558
C01162=13.550,-89.334,75.383,178.6906,-6.5704,-12771.3752
C01163=12.382,-82.740,74.428,179.8876,-6.7409,-12771.4889
C01164=11.418,-75.576,72.474,179.9164,-5.7880,-12771.4087
C01165=10.544,-69.129,69.894,179.8743,-4.3120,-12771.3277
C01166=9.686,-64.262,67.375,179.9289,-0.8741,-12771.4285
C01167=8.195,-61.417,65.554,-164.1096,17.3895,-12772.3998
C01168=4.967,-60.695,64.832,-145.5318,6.2395,-12775.3216
C01169=2.212,-60.785,64.801,-144.4407,-0.2926,-12777.9159
C01170=0.000,-60.820,64.822,-144.4503,-0.0000,-12780.0000
C01171=0.000,-60.820,64.822,-144.4503,-0.0000,-12780.0000
C01172=-2.212,-60.785,64.801,-144.4407,0.2926,-12782.0841
C01173=-4.967,-60.695,64.832,-145.5318,-6.2395,-12784.6784
C01174=-8.195,-61.417,65.554,-164.1096,-17.3895,-12787.6002
C01175=-9.686,-64.262,67.375,179.9289,0.8741,-12788.5715
C01176=-10.544,-69.129,69.894,179.8743,4.3120,-12788.6723
C01177=-11.418,-75.576,72.474,179.9164,5.7880,-12788.5913
C01178=-12.382,-82.740,74.428,179.8876,6.7409,-12788.5111
C01179=-13.550,-89.334,75.383,178.6906,6.5704,-12788.6248
C01180=-17.016,-94.154,75.883,177.1656,3.1658,-12790.2442
C01181=-22.407,-96.473,76.288,178.0701,0.7603,-12793.0758
C01182=-28.621,-95.791,76.696,179.8623,-0.0007,-12796.6354
C01183=-35.046,-93.654,76.964,179.9819,0.0007,-12800.5162
C01184=-41.442,-91.005,76.964,179.9820,0.0019,-12804.4836
C01185=-47.497,-87.973,76.696,179.8642,0.0017,-12808.3648
C01186=-52.372,-84.060,76.288,178.0752,-0.7593,-12811.9242
C01187=-54.545,-78.609,75.883,177.1688,-3.1633,-12814.7559
C01188=-53.588,-72.750,75.383,178.6911,-6.5728,-12816.3755
C01189=-49.751,-67.261,74.428,179.8915,-6.7417,-12816.4893
C01190=-45.367,-61.514,72.474,179.9177,-5.7873,-12816.4090
C01191=-41.426,-56.337,69.894,179.8743,-4.3140,-12816.3280
C01192=-38.591,-52.289,67.375,179.9265,-0.8715,-12816.4285
C01193=-37.634,-49.223,65.554,-164.1107,17.3872,-12817.4001
C01194=-39.406,-46.429,64.832,-145.5293,6.2383,-12820.3225
C01195=-41.417,-44.545,64.801,-144.4394,-0.2887,-12822.9160
C01196=-43.006,-43.006,64.822,-144.4511,0.0000,-12825.0000
C01197=-44.545,-41.417,64.801,-144.4394,0.2887,-12827.0840
C01198=-46.430,-39.405,64.832,-145.5330,-6.2436,-12829.6788
C01199=-49.223,-37.634,65.554,-164.1107,-17.3872,-12832.5999
C01200=-52.289,-38.591,67.375,179.9265,0.8715,-12833.5715
C01201=-56.337,-41.426,69.894,179.8743,4.3140,-12833.6720
C01202=-61.514,-45.367,72.474,179.9177,5.7873,-12833.5910
C01203=-67.261,-49.751,74.428,179.8915,6.7417,-12833.5107
C01204=-72.750,-53.588,75.383,178.6911,6.5728,-12833.6245
C01205=-78.609,-54.545,75.883,177.1688,3.1633,-12835.2441
C01206=-84.060,-52.372,76.288,178.0752,0.7593,-12838.0758
C01207=-87.973,-47.497,76.696,179.8642,-0.0017,-12841.6352
C01208=-91.005,-41.442,76.964,179.9820,-0.0019,-12845.5164
C01209=-93.654,-35.046,76.964,179.9819,-0.0007,-12849.4838
C01210=-95.791,-28.621,76.696,179.8623,0.0007,-12853.3646
C01211=-96.473,-22.407,76.288,178.0701,-0.7603,-12856.9242
C01212=-94.154,-17.016,75.883,177.1656,-3.1658,-12859.7558
C01213=-89.334,-13.550,75.383,178.6906,-6.5704,-12861.3752
C01214=-82.740,-12.382,74.428,179.8876,-6.7409,-12861.4889
C01215=-75.576,-11.418,72.474,179.9164,-5.7880,-12861.4087
C01216=-69.129,-10.544,69.894,179.8743,-4.3120,-12861.3277
C01217=-64.262,-9.686,67.375,179.9289,-0.8741,-12861.4285
C01218=-61.417,-8.195,65.554,-164.1096,17.3895,-12862.3998
C01219=-60.695,-4.967,64.832,-145.5318,6.2395,-12865.3216
C01220=-60.785,-2.212,64.801,-144.4407,-0.2926,-12867.9159
C01221=-60.820,0.000,64.822,-144.4503,0.0000,-12870.0000
C01222=-60.785,2.212,64.801,-144.4407,0.2926,-12872.0841
C01223=-60.695,4.967,64.832,-145.5318,-6.2395,-12874.6784
C01224=-61.417,8.195,65.554,-164.1096,-17.3895,-12877.6002
C01225=-64.262,9.686,67.375,179.9289,0.8741,-12878.5715
C01226=-69.129,10.544,69.894,179.8743,4.3120,-12878.6723
C01227=-75.576,11.418,72.474,179.9164,5.7880,-12878.5913
C01228=-82.740,12.382,74.428,179.8876,6.7409,-12878.5111
C01229=-89.334,13.550,75.383,178.6906,6.5704,-12878.6248
C01230=-94.154,17.016,75.883,177.1656,3.1658,-12880.2442
C01231=-96.473,22.407,76.288,178.0701,0.7603,-12883.0758
C01232=-95.791,28.621,76.696,179.8623,-0.0007,-12886.6354
C01233=-93.654,35.046,76.964,179.9819,0.0007,-12890.5162
C01234=-91.005,41.442,76.964,179.9820,0.0019,-12894.4836
C01235=-87.973,47.497,76.696,179.8642,0.0017,-12898.3648
C01236=-84.060,52.372,76.288,178.0752,-0.7593,-12901.9242
C01237=-78.609,54.545,75.883,177.1688,-3.1633,-12904.7559
C01238=-72.750,53.588,75.383,178.6911,-6.5728,-12906.3755
C01239=-67.261,49.751,74.428,179.8915,-6.7417,-12906.4893
C01240=-61.514,45.367,72.474,179.9177,-5.7873,-12906.4090
C01241=-56.337,41.426,69.894,179.8743,-4.3140,-12906.3280
C01242=-52.289,38.591,67.375,179.9265,-0.8715,-12906.4285
C01243=-49.223,37.634,65.554,-164.1107,17.3872,-12907.4001
C01244=-46.429,39.406,64.832,-145.5293,6.2383,-12910.3225
C01245=-44.545,41.417,64.801,-144.4394,-0.2887,-12912.9160
C01246=-43.006,43.006,64.822,-144.4511,0.0000,-12915.0000
C01247=-41.417,44.545,64.801,-144.4394,0.2887,-12917.0840
C01248=-39.405,46.430,64.832,-145.5330,-6.2436,-12919.6788
C01249=-37.634,49.223,65.554,-164.1107,-17.3872,-12922.5999
C01250=-38.591,52.289,67.375,179.9265,0.8715,-12923.5715
C01251=-41.426,56.337,69.894,179.8743,4.3140,-12923.6720
C01252=-45.367,61.514,72.474,179.9177,5.7873,-12923.5910
C01253=-49.751,67.261,74.428,179.8915,6.7417,-12923.5107
C01254=-53.588,72.750,75.383,178.6911,6.5728,-12923.6245
C01255=-54.545,78.609,75.883,177.1688,3.1633,-12925.2441
C01256=-52.372,84.060,76.288,178.0752,0.7593,-12928.0758
C01257=-47.497,87.973,76.696,179.8642,-0.0017,-12931.6352
C01258=-41.442,91.005,76.964,179.9820,-0.0019,-12935.5164
C01259=-35.046,93.654,76.964,179.9819,-0.0007,-12939.4838
C01260=-28.621,95.791,76.696,179.8623,0.0007,-12943.3646
C01261=-22.407,96.473,76.288,178.0701,-0.7603,-12946.9242
C01262=-17.016,94.154,75.883,177.1656,-3.1658,-12949.7558
C01263=-13.550,89.334,75.383,178.6906,-6.5704,-12951.3752
C01264=-12.382,82.740,74.428,179.8876,-6.7409,-12951.4889
C01265=-11.418,75.576,72.474,179.9164,-5.7880,-12951.4087
C01266=-10.544,69.129,69.894,179.8743,-4.3120,-12951.3277
C01267=-9.686,64.262,67.375,179.9289,-0.8741,-12951.4285
C01268=-8.195,61.417,65.554,-164.1096,17.3895,-12952.3998
C01269=-4.967,60.695,64.832,-145.5318,6.2395,-12955.3216
C01270=-2.212,60.785,64.801,-144.4407,-0.2926,-12957.9159
C01271=0.000,60.820,64.822,-144.4503,0.0000,-12960.0000
C01272=0.000,59.554,66.621,-145.3422,0.0000,-12960.0000
C01273=2.097,59.523,66.599,-145.3345,0.2770,-12962.0177
C01274=4.772,59.445,66.632,-146.5013,-6.3202,-12964.5896
C01275=7.959,60.221,67.386,-165.4665,-16.6506,-12967.5288
C01276=9.406,63.206,69.285,179.9095,1.2996,-12968.4644
C01277=10.239,68.282,71.901,179.9006,4.2888,-12968.5281
C01278=11.109,74.974,74.567,179.9369,5.5259,-12968.4283
C01279=12.073,82.372,76.575,179.9220,6.3189,-12968.3383
C01280=13.226,89.158,77.551,178.8203,6.1239,-12968.4379
C01281=16.717,94.118,78.062,177.3801,2.9713,-12970.0717
C01282=22.174,96.515,78.476,178.2110,0.7111,-12972.9390
C01283=28.477,95.839,78.891,179.8749,0.0013,-12976.5485
C01284=34.998,93.673,79.163,179.9873,-0.0014,-12980.4866
C01285=41.489,90.984,79.163,179.9872,-0.0005,-12984.5131
C01286=47.632,87.904,78.891,179.8743,-0.0035,-12988.4517
C01287=52.567,83.926,78.476,178.2090,-0.7111,-12992.0609
C01288=54.731,78.373,78.062,177.3787,-2.9711,-12994.9281
C01289=53.692,72.396,77.551,178.8240,-6.1292,-12996.5622
C01290=49.709,66.782,76.575,179.9204,-6.3181,-12996.6621
C01291=45.159,60.870,74.567,179.9368,-5.5263,-12996.5714
C01292=41.042,55.523,71.901,179.8966,-4.2883,-12996.4714
C01293=38.042,51.344,69.285,179.9067,-1.3002,-12996.5356
C01294=36.955,48.211,67.386,-165.4649,16.6464,-12997.4711
C01295=38.660,45.408,66.632,-146.5038,6.3217,-13000.4108
C01296=40.607,43.572,66.599,-145.3345,-0.2753,-13002.9827
C01297=42.111,42.111,66.621,-145.3443,0.0000,-13005.0000
C01298=43.571,40.607,66.599,-145.3311,0.2805,-13007.0166
C01299=45.409,38.659,66.632,-146.5039,-6.3225,-13009.5906
C01300=48.211,36.955,67.386,-165.4695,-16.6499,-13012.5289
C01301=51.344,38.042,69.285,179.9067,1.3002,-13013.4644
C01302=55.523,41.042,71.901,179.8966,4.2883,-13013.5286
C01303=60.870,45.159,74.567,179.9368,5.5263,-13013.4286
C01304=66.782,49.709,76.575,179.9204,6.3181,-13013.3379
C01305=72.396,53.692,77.551,178.8240,6.1292,-13013.4378
C01306=78.373,54.731,78.062,177.3787,2.9711,-13015.0719
C01307=83.926,52.567,78.476,178.2090,0.7111,-13017.9391
C01308=87.904,47.632,78.891,179.8743,0.0035,-13021.5483
C01309=90.984,41.489,79.163,179.9872,0.0005,-13025.4869
C01310=93.673,34.998,79.163,179.9873,0.0014,-13029.5134
C01311=95.839,28.477,78.891,179.8749,-0.0013,-13033.4515
C01312=96.515,22.174,78.476,178.2110,-0.7111,-13037.0610
C01313=94.118,16.717,78.062,177.3801,-2.9713,-13039.9283
C01314=89.158,13.226,77.551,178.8203,-6.1239,-13041.5621
C01315=82.372,12.073,76.575,179.9220,-6.3189,-13041.6617
C01316=74.974,11.109,74.567,179.9369,-5.5259,-13041.5717
C01317=68.282,10.239,71.901,179.9006,-4.2888,-13041.4719
C01318=63.206,9.406,69.285,179.9095,-1.2996,-13041.5356
C01319=60.221,7.959,67.386,-165.4665,16.6506,-13042.4712
C01320=59.445,4.772,66.632,-146.5013,6.3202,-13045.4104
C01321=59.523,2.097,66.599,-145.3345,-0.2770,-13047.9823
C01322=59.554,0.000,66.621,-145.3422,0.0000,-13050.0000
C01323=59.523,-2.096,66.599,-145.3345,0.2777,-13052.0167
C01324=59.445,-4.772,66.632,-146.5061,-6.3197,-13054.5896
C01325=60.222,-7.959,67.386,-165.4665,-16.6506,-13057.5286
C01326=63.206,-9.406,69.285,179.9095,1.2996,-13058.4644
C01327=68.282,-10.239,71.901,179.9006,4.2888,-13058.5281
C01328=74.974,-11.109,74.567,179.9369,5.5259,-13058.4283
C01329=82.372,-12.073,76.575,179.9220,6.3189,-13058.3383
C01330=89.158,-13.226,77.551,178.8203,6.1239,-13058.4379
C01331=94.118,-16.717,78.062,177.3801,2.9713,-13060.0717
C01332=96.515,-22.174,78.476,178.2110,0.7111,-13062.9390
C01333=95.839,-28.477,78.891,179.8749,0.0013,-13066.5485
C01334=93.673,-34.998,79.163,179.9873,-0.0014,-13070.4866
C01335=90.984,-41.489,79.163,179.9872,-0.0005,-13074.5131
C01336=87.904,-47.632,78.891,179.8743,-0.0035,-13078.4517
C01337=83.926,-52.567,78.476,178.2090,-0.7111,-13082.0609
C01338=78.373,-54.731,78.062,177.3787,-2.9711,-13084.9281
C01339=72.396,-53.692,77.551,178.8240,-6.1292,-13086.5622
C01340=66.782,-49.709,76.575,179.9204,-6.3181,-13086.6621
C01341=60.870,-45.159,74.567,179.9368,-5.5263,-13086.5714
C01342=55.523,-41.042,71.901,179.8966,-4.2883,-13086.4714
C01343=51.344,-38.042,69.285,179.9067,-1.3002,-13086.5356
C01344=48.211,-36.955,67.386,-165.4649,16.6464,-13087.4711
C01345=45.408,-38.660,66.632,-146.5038,6.3217,-13090.4108
C01346=43.572,-40.607,66.599,-145.3345,-0.2753,-13092.9827
C01347=42.111,-42.111,66.621,-145.3443,0.0000,-13095.0000
C01348=40.607,-43.571,66.599,-145.3311,0.2805,-13097.0166
C01349=38.659,-45.409,66.632,-146.5039,-6.3225,-13099.5906
C01350=36.955,-48.211,67.386,-165.4695,-16.6499,-13102.5289
C01351=38.042,-51.344,69.285,179.9067,1.3002,-13103.4644
C01352=41.042,-55.523,71.901,179.8966,4.2883,-13103.5286
C01353=45.159,-60.870,74.567,179.9368,5.5263,-13103.4286
C01354=49.709,-66.782,76.575,179.9204,6.3181,-13103.3379
C01355=53.692,-72.396,77.551,178.8240,6.1292,-13103.4378
C01356=54.731,-78.373,78.062,177.3787,2.9711,-13105.0719
C01357=52.567,-83.926,78.476,178.2090,0.7111,-13107.9391
C01358=47.632,-87.904,78.891,179.8743,0.0035,-13111.5483
C01359=41.489,-90.984,79.163,179.9872,0.0005,-13115.4869
C01360=34.998,-93.673,79.163,179.9873,0.0014,-13119.5134
C01361=28.477,-95.839,78.891,179.8749,-0.0013,-13123.4515
C01362=22.174,-96.515,78.476,178.2110,-0.7111,-13127.0610
C01363=16.717,-94.118,78.062,177.3801,-2.9713,-13129.9283
C01364=13.226,-89.158,77.551,178.8203,-6.1239,-13131.5621
C01365=12.073,-82.372,76.575,179.9220,-6.3189,-13131.6617
C01366=11.109,-74.974,74.567,179.9369,-5.5259,-13131.5717
C01367=10.239,-68.282,71.901,179.9006,-4.2888,-13131.4719
C01368=9.406,-63.206,69.285,179.9095,-1.2996,-13131.5356
C01369=7.959,-60.221,67.386,-165.4665,16.6506,-13132.4712
C01370=4.772,-59.445,66.632,-146.5013,6.3202,-13135.4104
C01371=2.097,-59.523,66.599,-145.3345,-0.2770,-13137.9823
C01372=0.000,-59.554,66.621,-145.3422,-0.0000,-13140.0000
C01373=0.000,-59.554,66.621,-145.3422,-0.0000,-13140.0000
C01374=-2.096,-59.523,66.599,-145.3345,0.2777,-13142.0167
C01375=-4.772,-59.445,66.632,-146.5061,-6.3197,-13144.5896
C01376=-7.959,-60.222,67.386,-165.4665,-16.6506,-13147.5286
C01377=-9.406,-63.206,69.285,179.9095,1.2996,-13148.4644
C01378=-10.239,-68.282,71.901,179.9006,4.2888,-13148.5281
C01379=-11.109,-74.974,74.567,179.9369,5.5259,-13148.4283
C01380=-12.073,-82.372,76.575,179.9220,6.3189,-13148.3383
C01381=-13.226,-89.158,77.551,178.8203,6.1239,-13148.4379
C01382=-16.717,-94.118,78.062,177.3801,2.9713,-13150.0717
C01383=-22.174,-96.515,78.476,178.2110,0.7111,-13152.9390
C01384=-28.477,-95.839,78.891,179.8749,0.0013,-13156.5485
C01385=-34.998,-93.673,79.163,179.9873,-0.0014,-13160.4866
C01386=-41.489,-90.984,79.163,179.9872,-0.0005,-13164.5131
C01387=-47.632,-87.904,78.891,179.8743,-0.0035,-13168.4517
C01388=-52.567,-83.926,78.476,178.2090,-0.7111,-13172.0609
C01389=-54.731,-78.373,78.062,177.3787,-2.9711,-13174.9281
C01390=-53.692,-72.396,77.551,178.8240,-6.1292,-13176.5622
C01391=-49.709,-66.782,76.575,179.9204,-6.3181,-13176.6621
C01392=-45.159,-60.870,74.567,179.9368,-5.5263,-13176.5714
C01393=-41.042,-55.523,71.901,179.8966,-4.2883,-13176.4714
C01394=-38.042,-51.344,69.285,179.9067,-1.3002,-13176.5356
C01395=-36.955,-48.211,67.386,-165.4649,16.6464,-13177.4711
C01396=-38.660,-45.408,66.632,-146.5038,6.3217,-13180.4108
C01397=-40.607,-43.572,66.599,-145.3345,-0.2753,-13182.9827
C01398=-42.111,-42.111,66.621,-145.3443,-0.0000,-13185.0000
C01399=-43.571,-40.607,66.599,-145.3311,0.2805,-13187.0166
C01400=-45.409,-38.659,66.632,-146.5039,-6.3225,-13189.5906
C01401=-48.211,-36.955,67.386,-165.4695,-16.6499,-13192.5289
C01402=-51.344,-38.042,69.285,179.9067,1.3002,-13193.4644
C01403=-55.523,-41.042,71.901,179.8966,4.2883,-13193.5286
C01404=-60.870,-45.159,74.567,179.9368,5.5263,-13193.4286
C01405=-66.782,-49.709,76.575,179.9204,6.3181,-13193.3379
C01406=-72.396,-53.692,77.551,178.8240,6.1292,-13193.4378
C01407=-78.373,-54.731,78.062,177.3787,2.9711,-13195.0719
C01408=-83.926,-52.567,78.476,178.2090,0.7111,-13197.9391
C01409=-87.904,-47.632,78.891,179.8743,0.0035,-13201.5483
C01410=-90.984,-41.489,79.163,179.9872,0.0005,-13205.4869
C01411=-93.673,-34.998,79.163,179.9873,0.0014,-13209.5134
C01412=-95.839,-28.477,78.891,179.8749,-0.0013,-13213.4515
C01413=-96.515,-22.174,78.476,178.2110,-0.7111,-13217.0610
C01414=-94.118,-16.717,78.062,177.3801,-2.9713,-13219.9283
C01415=-89.158,-13.226,77.551,178.8203,-6.1239,-13221.5621
C01416=-82.372,-12.073,76.575,179.9220,-6.3189,-13221.6617
C01417=-74.974,-11.109,74.567,179.9369,-5.5259,-13221.5717
C01418=-68.282,-10.239,71.901,179.9006,-4.2888,-13221.4719
C01419=-63.206,-9.406,69.285,179.9095,-1.2996,-13221.5356
C01420=-60.221,-7.959,67.386,-165.4665,16.6506,-13222.4712
C01421=-59.445,-4.772,66.632,-146.5013,6.3202,-13225.4104
C01422=-59.523,-2.097,66.599,-145.3345,-0.2770,-13227.9823
C01423=-59.554,0.000,66.621,-145.3422,-0.0000,-13230.0000
C01424=-59.523,2.096,66.599,-145.3345,0.2777,-13232.0167
C01425=-59.445,4.772,66.632,-146.5061,-6.3197,-13234.5896
C01426=-60.222,7.959,67.386,-165.4665,-16.6506,-13237.5286
C01427=-63.206,9.406,69.285,179.9095,1.2996,-13238.4644
C01428=-68.282,10.239,71.901,179.9006,4.2888,-13238.5281
C01429=-74.974,11.109,74.567,179.9369,5.5259,-13238.4283
C01430=-82.372,12.073,76.575,179.9220,6.3189,-13238.3383
C01431=-89.158,13.226,77.551,178.8203,6.1239,-13238.4379
C01432=-94.118,16.717,78.062,177.3801,2.9713,-13240.0717
C01433=-96.515,22.174,78.476,178.2110,0.7111,-13242.9390
C01434=-95.839,28.477,78.891,179.8749,0.0013,-13246.5485
C01435=-93.673,34.998,79.163,179.9873,-0.0014,-13250.4866
C01436=-90.984,41.489,79.163,179.9872,-0.0005,-13254.5131
C01437=-87.904,47.632,78.891,179.8743,-0.0035,-13258.4517
C01438=-83.926,52.567,78.476,178.2090,-0.7111,-13262.0609
C01439=-78.373,54.731,78.062,177.3787,-2.9711,-13264.9281
C01440=-72.396,53.692,77.551,178.8240,-6.1292,-13266.5622
C01441=-66.782,49.709,76.575,179.9204,-6.3181,-13266.6621
C01442=-60.870,45.159,74.567,179.9368,-5.5263,-13266.5714
C01443=-55.523,41.042,71.901,179.8966,-4.2883,-13266.4714
C01444=-51.344,38.042,69.285,179.9067,-1.3002,-13266.5356
C01445=-48.211,36.955,67.386,-165.4649,16.6464,-13267.4711
C01446=-45.408,38.660,66.632,-146.5038,6.3217,-13270.4108
C01447=-43.572,40.607,66.599,-145.3345,-0.2753,-13272.9827
C01448=-42.111,42.111,66.621,-145.3443,-0.0000,-13275.0000
C01449=-40.607,43.571,66.599,-145.3311,0.2805,-13277.0166
C01450=-38.659,45.409,66.632,-146.5039,-6.3225,-13279.5906
C01451=-36.955,48.211,67.386,-165.4695,-16.6499,-13282.5289
C01452=-38.042,51.344,69.285,179.9067,1.3002,-13283.4644
C01453=-41.042,55.523,71.901,179.8966,4.2883,-13283.5286
C01454=-45.159,60.870,74.567,179.9368,5.5263,-13283.4286
C01455=-49.709,66.782,76.575,179.9204,6.3181,-13283.3379
C01456=-53.692,72.396,77.551,178.8240,6.1292,-13283.4378
C01457=-54.731,78.373,78.062,177.3787,2.9711,-13285.0719
C01458=-52.567,83.926,78.476,178.2090,0.7111,-13287.9391
C01459=-47.632,87.904,78.891,179.8743,0.0035,-13291.5483
C01460=-41.489,90.984,79.163,179.9872,0.0005,-13295.4869
C01461=-34.998,93.673,79.163,179.9873,0.0014,-13299.5134
C01462=-28.477,95.839,78.891,179.8749,-0.0013,-13303.4515
C01463=-22.174,96.515,78.476,178.2110,-0.7111,-13307.0610
C01464=-16.717,94.118,78.062,177.3801,-2.9713,-13309.9283
C01465=-13.226,89.158,77.551,178.8203,-6.1239,-13311.5621
C01466=-12.073,82.372,76.575,179.9220,-6.3189,-13311.6617
C01467=-11.109,74.974,74.567,179.9369,-5.5259,-13311.5717
C01468=-10.239,68.282,71.901,179.9006,-4.2888,-13311.4719
C01469=-9.406,63.206,69.285,179.9095,-1.2996,-13311.5356
C01470=-7.959,60.222,67.386,-165.4665,16.6506,-13312.4714
C01471=-4.772,59.445,66.632,-146.5061,6.3197,-13315.4104
C01472=-2.096,59.523,66.599,-145.3345,-0.2777,-13317.9833
C01473=0.000,59.554,66.621,-145.3422,0.0000,-13320.0000
C01474=0.000,58.319,68.442,-146.3576,0.0000,-13320.0000
C01475=1.984,58.291,68.419,-146.3472,0.2651,-13321.9494
C01476=4.582,58.225,68.453,-147.5982,-6.3565,-13324.4996
C01477=7.730,59.058,69.238,-166.7870,-15.8213,-13327.4570
C01478=9.135,62.185,71.215,179.8995,1.6423,-13328.3570
C01479=9.949,67.473,73.927,179.9174,4.1975,-13328.3879
C01480=10.820,74.409,76.674,179.9569,5.2067,-13328.2735
C01481=11.787,82.032,78.729,179.9453,5.8354,-13328.1767
C01482=12.929,88.996,79.725,178.9564,5.6149,-13328.2659
C01483=16.445,94.085,80.245,177.6180,2.7341,-13329.9145
C01484=21.964,96.553,80.665,178.3734,0.6523,-13332.8156
C01485=28.347,95.882,81.086,179.8859,-0.0021,-13336.4700
C01486=34.955,93.690,81.363,179.9873,-0.0014,-13340.4601
C01487=41.532,90.965,81.363,179.9872,-0.0005,-13344.5401
C01488=47.755,87.843,81.086,179.8820,-0.0011,-13348.5303
C01489=52.743,83.804,80.665,178.3730,-0.6487,-13352.1847
C01490=54.900,78.157,80.245,177.6189,-2.7304,-13355.0854
C01491=53.787,72.072,79.725,178.9551,-5.6184,-13356.7338
C01492=49.670,66.340,78.729,179.9437,-5.8304,-13356.8229
C01493=44.964,60.266,76.674,179.9532,-5.2050,-13356.7263
C01494=40.676,54.746,73.927,179.9178,-4.1971,-13356.6122
C01495=37.512,50.430,71.215,179.9010,-1.6404,-13356.6435
C01496=36.294,47.226,69.238,-166.7829,15.8226,-13357.5429
C01497=37.931,44.411,68.453,-147.5962,6.3553,-13360.5003
C01498=39.816,42.621,68.419,-146.3455,-0.2653,-13363.0512
C01499=41.238,41.238,68.442,-146.3534,0.0000,-13365.0000
C01500=42.621,39.816,68.419,-146.3455,0.2653,-13366.9488
C01501=44.412,37.931,68.453,-147.6000,-6.3600,-13369.5003
C01502=47.226,36.294,69.238,-166.7829,-15.8226,-13372.4571
C01503=50.430,37.512,71.215,179.9010,1.6404,-13373.3565
C01504=54.746,40.676,73.927,179.9178,4.1971,-13373.3878
C01505=60.266,44.964,76.674,179.9532,5.2050,-13373.2737
C01506=66.340,49.670,78.729,179.9437,5.8304,-13373.1771
C01507=72.072,53.787,79.725,178.9551,5.6184,-13373.2662
C01508=78.157,54.900,80.245,177.6189,2.7304,-13374.9146
C01509=83.804,52.743,80.665,178.3730,0.6487,-13377.8153
C01510=87.843,47.755,81.086,179.8820,0.0011,-13381.4697
C01511=90.965,41.532,81.363,179.9872,0.0005,-13385.4599
C01512=93.690,34.955,81.363,179.9873,0.0014,-13389.5399
C01513=95.882,28.347,81.086,179.8859,0.0021,-13393.5300
C01514=96.553,21.964,80.665,178.3734,-0.6523,-13397.1844
C01515=94.085,16.445,80.245,177.6180,-2.7341,-13400.0855
C01516=88.996,12.929,79.725,178.9564,-5.6149,-13401.7341
C01517=82.032,11.787,78.729,179.9453,-5.8354,-13401.8233
C01518=74.409,10.820,76.674,179.9569,-5.2067,-13401.7265
C01519=67.473,9.949,73.927,179.9174,-4.1975,-13401.6121
C01520=62.185,9.135,71.215,179.8995,-1.6423,-13401.6430
C01521=59.058,7.730,69.238,-166.7870,15.8213,-13402.5430
C01522=58.225,4.582,68.453,-147.5982,6.3565,-13405.5004
C01523=58.291,1.984,68.419,-146.3472,-0.2651,-13408.0506
C01524=58.319,0.000,68.442,-146.3576,0.0000,-13410.0000
C01525=58.291,-1.983,68.419,-146.3472,0.2658,-13411.9484
C01526=58.225,-4.583,68.453,-147.5983,-6.3571,-13414.5006
C01527=59.058,-7.730,69.238,-166.7870,-15.8213,-13417.4570
C01528=62.185,-9.135,71.215,179.8995,1.6423,-13418.3570
C01529=67.473,-9.949,73.927,179.9174,4.1975,-13418.3879
C01530=74.409,-10.820,76.674,179.9569,5.2067,-13418.2735
C01531=82.032,-11.787,78.729,179.9453,5.8354,-13418.1767
C01532=88.996,-12.929,79.725,178.9564,5.6149,-13418.2659
C01533=94.085,-16.445,80.245,177.6180,2.7341,-13419.9145
C01534=96.553,-21.964,80.665,178.3734,0.6523,-13422.8156
C01535=95.882,-28.347,81.086,179.8859,-0.0021,-13426.4700
C01536=93.690,-34.955,81.363,179.9873,-0.0014,-13430.4601
C01537=90.965,-41.532,81.363,179.9872,-0.0005,-13434.5401
C01538=87.843,-47.755,81.086,179.8820,-0.0011,-13438.5303
C01539=83.804,-52.743,80.665,178.3730,-0.6487,-13442.1847
C01540=78.157,-54.900,80.245,177.6189,-2.7304,-13445.0854
C01541=72.072,-53.787,79.725,178.9551,-5.6184,-13446.7338
C01542=66.340,-49.670,78.729,179.9437,-5.8304,-13446.8229
C01543=60.266,-44.964,76.674,179.9532,-5.2050,-13446.7263
C01544=54.746,-40.676,73.927,179.9178,-4.1971,-13446.6122
C01545=50.430,-37.512,71.215,179.9010,-1.6404,-13446.6435
C01546=47.226,-36.294,69.238,-166.7829,15.8226,-13447.5429
C01547=44.411,-37.931,68.453,-147.5962,6.3553,-13450.5003
C01548=42.621,-39.816,68.419,-146.3455,-0.2653,-13453.0512
C01549=41.238,-41.238,68.442,-146.3534,0.0000,-13455.0000
C01550=39.816,-42.621,68.419,-146.3455,0.2653,-13456.9488
C01551=37.931,-44.412,68.453,-147.6000,-6.3600,-13459.5003
C01552=36.294,-47.226,69.238,-166.7829,-15.8226,-13462.4571
C01553=37.512,-50.430,71.215,179.9010,1.6404,-13463.3565
C01554=40.676,-54.746,73.927,179.9178,4.1971,-13463.3878
C01555=44.964,-60.266,76.674,179.9532,5.2050,-13463.2737
C01556=49.670,-66.340,78.729,179.9437,5.8304,-13463.1771
C01557=53.787,-72.072,79.725,178.9551,5.6184,-13463.2662
C01558=54.900,-78.157,80.245,177.6189,2.7304,-13464.9146
C01559=52.743,-83.804,80.665,178.3730,0.6487,-13467.8153
C01560=47.755,-87.843,81.086,179.8820,0.0011,-13471.4697
C01561=41.532,-90.965,81.363,179.9872,0.0005,-13475.4599
C01562=34.955,-93.690,81.363,179.9873,0.0014,-13479.5399
C01563=28.347,-95.882,81.086,179.8859,0.0021,-13483.5300
C01564=21.964,-96.553,80.665,178.3734,-0.6523,-13487.1844
C01565=16.445,-94.085,80.245,177.6180,-2.7341,-13490.0855
C01566=12.929,-88.996,79.725,178.9564,-5.6149,-13491.7341
C01567=11.787,-82.032,78.729,179.9453,-5.8354,-13491.8233
C01568=10.820,-74.409,76.674,179.9569,-5.2067,-13491.7265
C01569=9.949,-67.473,73.927,179.9174,-4.1975,-13491.6121
C01570=9.135,-62.185,71.215,179.8995,-1.6423,-13491.6430
C01571=7.730,-59.058,69.238,-166.7870,15.8213,-13492.5430
C01572=4.582,-58.225,68.453,-147.5982,6.3565,-13495.5004
C01573=1.984,-58.291,68.419,-146.3472,-0.2651,-13498.0506
C01574=0.000,-58.319,68.442,-146.3576,0.0000,-13500.0000
C01575=0.000,-58.319,68.442,-146.3576,0.0000,-13500.0000
C01576=-1.983,-58.291,68.419,-146.3472,0.2658,-13501.9484
C01577=-4.583,-58.225,68.453,-147.5983,-6.3571,-13504.5006
C01578=-7.730,-59.058,69.238,-166.7870,-15.8213,-13507.4570
C01579=-9.135,-62.185,71.215,179.8995,1.6423,-13508.3570
C01580=-9.949,-67.473,73.927,179.9174,4.1975,-13508.3879
C01581=-10.820,-74.409,76.674,179.9569,5.2067,-13508.2735
C01582=-11.787,-82.032,78.729,179.9453,5.8354,-13508.1767
C01583=-12.929,-88.996,79.725,178.9564,5.6149,-13508.2659
C01584=-16.445,-94.085,80.245,177.6180,2.7341,-13509.9145
C01585=-21.964,-96.553,80.665,178.3734,0.6523,-13512.8156
C01586=-28.347,-95.882,81.086,179.8859,-0.0021,-13516.4700
C01587=-34.955,-93.690,81.363,179.9873,-0.0014,-13520.4601
C01588=-41.532,-90.965,81.363,179.9872,-0.0005,-13524.5401
C01589=-47.755,-87.843,81.086,179.8820,-0.0011,-13528.5303
C01590=-52.743,-83.804,80.665,178.3730,-0.6487,-13532.1847
C01591=-54.900,-78.157,80.245,177.6189,-2.7304,-13535.0854
C01592=-53.787,-72.072,79.725,178.9551,-5.6184,-13536.7338
C01593=-49.670,-66.340,78.729,179.9437,-5.8304,-13536.8229
C01594=-44.964,-60.266,76.674,179.9532,-5.2050,-13536.7263
C01595=-40.676,-54.746,73.927,179.9178,-4.1971,-13536.6122
C01596=-37.512,-50.430,71.215,179.9010,-1.6404,-13536.6435
C01597=-36.294,-47.226,69.238,-166.7829,15.8226,-13537.5429
C01598=-37.931,-44.411,68.453,-147.5962,6.3553,-13540.5003
C01599=-39.816,-42.621,68.419,-146.3455,-0.2653,-13543.0512
C01600=-41.238,-41.238,68.442,-146.3534,0.0000,-13545.0000
C01601=-42.621,-39.816,68.419,-146.3455,0.2653,-13546.9488
C01602=-44.412,-37.931,68.453,-147.6000,-6.3600,-13549.5003
C01603=-47.226,-36.294,69.238,-166.7829,-15.8226,-13552.4571
C01604=-50.430,-37.512,71.215,179.9010,1.6404,-13553.3565
C01605=-54.746,-40.676,73.927,179.9178,4.1971,-13553.3878
C01606=-60.266,-44.964,76.674,179.9532,5.2050,-13553.2737
C01607=-66.340,-49.670,78.729,179.9437,5.8304,-13553.1771
C01608=-72.072,-53.787,79.725,178.9551,5.6184,-13553.2662
C01609=-78.157,-54.900,80.245,177.6189,2.7304,-13554.9146
C01610=-83.804,-52.743,80.665,178.3730,0.6487,-13557.8153
C01611=-87.843,-47.755,81.086,179.8820,0.0011,-13561.4697
C01612=-90.965,-41.532,81.363,179.9872,0.0005,-13565.4599
C01613=-93.690,-34.955,81.363,179.9873,0.0014,-13569.5399
C01614=-95.882,-28.347,81.086,179.8859,0.0021,-13573.5300
C01615=-96.553,-21.964,80.665,178.3734,-0.6523,-13577.1844
C01616=-94.085,-16.445,80.245,177.6180,-2.7341,-13580.0855
C01617=-88.996,-12.929,79.725,178.9564,-5.6149,-13581.7341
C01618=-82.032,-11.787,78.729,179.9453,-5.8354,-13581.8233
C01619=-74.409,-10.820,76.674,179.9569,-5.2067,-13581.7265
C01620=-67.473,-9.949,73.927,179.9174,-4.1975,-13581.6121
C01621=-62.185,-9.135,71.215,179.8995,-1.6423,-13581.6430
C01622=-59.058,-7.730,69.238,-166.7870,15.8213,-13582.5430
C01623=-58.225,-4.582,68.453,-147.5982,6.3565,-13585.5004
C01624=-58.291,-1.984,68.419,-146.3472,-0.2651,-13588.0506
C01625=-58.319,0.000,68.442,-146.3576,0.0000,-13590.0000
C01626=-58.291,1.983,68.419,-146.3472,0.2658,-13591.9484
C01627=-58.225,4.583,68.453,-147.5983,-6.3571,-13594.5006
C01628=-59.058,7.730,69.238,-166.7870,-15.8213,-13597.4570
C01629=-62.185,9.135,71.215,179.8995,1.6423,-13598.3570
C01630=-67.473,9.949,73.927,179.9174,4.1975,-13598.3879
C01631=-74.409,10.820,76.674,179.9569,5.2067,-13598.2735
C01632=-82.032,11.787,78.729,179.9453,5.8354,-13598.1767
C01633=-88.996,12.929,79.725,178.9564,5.6149,-13598.2659
C01634=-94.085,16.445,80.245,177.6180,2.7341,-13599.9145
C01635=-96.553,21.964,80.665,178.3734,0.6523,-13602.8156
C01636=-95.882,28.347,81.086,179.8859,-0.0021,-13606.4700
C01637=-93.690,34.955,81.363,179.9873,-0.0014,-13610.4601
C01638=-90.965,41.532,81.363,179.9872,-0.0005,-13614.5401
C01639=-87.843,47.755,81.086,179.8820,-0.0011,-13618.5303
C01640=-83.804,52.743,80.665,178.3730,-0.6487,-13622.1847
C01641=-78.157,54.900,80.245,177.6189,-2.7304,-13625.0854
C01642=-72.072,53.787,79.725,178.9551,-5.6184,-13626.7338
C01643=-66.340,49.670,78.729,179.9437,-5.8304,-13626.8229
C01644=-60.266,44.964,76.674,179.9532,-5.2050,-13626.7263
C01645=-54.746,40.676,73.927,179.9178,-4.1971,-13626.6122
C01646=-50.430,37.512,71.215,179.9010,-1.6404,-13626.6435
C01647=-47.226,36.294,69.238,-166.7829,15.8226,-13627.5429
C01648=-44.411,37.931,68.453,-147.5962,6.3553,-13630.5003
C01649=-42.621,39.816,68.419,-146.3455,-0.2653,-13633.0512
C01650=-41.238,41.238,68.442,-146.3534,-0.0000,-13635.0000
C01651=-39.816,42.621,68.419,-146.3455,0.2653,-13636.9488
C01652=-37.931,44.412,68.453,-147.6000,-6.3600,-13639.5003
C01653=-36.294,47.226,69.238,-166.7829,-15.8226,-13642.4571
C01654=-37.512,50.430,71.215,179.9010,1.6404,-13643.3565
C01655=-40.676,54.746,73.927,179.9178,4.1971,-13643.3878
C01656=-44.964,60.266,76.674,179.9532,5.2050,-13643.2737
C01657=-49.670,66.340,78.729,179.9437,5.8304,-13643.1771
C01658=-53.787,72.072,79.725,178.9551,5.6184,-13643.2662
C01659=-54.900,78.157,80.245,177.6189,2.7304,-13644.9146
C01660=-52.743,83.804,80.665,178.3730,0.6487,-13647.8153
C01661=-47.755,87.843,81.086,179.8820,0.0011,-13651.4697
C01662=-41.532,90.965,81.363,179.9872,0.0005,-13655.4599
C01663=-34.955,93.690,81.363,179.9873,0.0014,-13659.5399
C01664=-28.347,95.882,81.086,179.8859,0.0021,-13663.5300
C01665=-21.964,96.553,80.665,178.3734,-0.6523,-13667.1844
C01666=-16.445,94.085,80.245,177.6180,-2.7341,-13670.0855
C01667=-12.929,88.996,79.725,178.9564,-5.6149,-13671.7341
C01668=-11.787,82.032,78.729,179.9453,-5.8354,-13671.8233
C01669=-10.820,74.409,76.674,179.9569,-5.2067,-13671.7265
C01670=-9.949,67.473,73.927,179.9174,-4.1975,-13671.6121
C01671=-9.135,62.185,71.215,179.8995,-1.6423,-13671.6430
C01672=-7.730,59.058,69.238,-166.7870,15.8213,-13672.5430
C01673=-4.583,58.225,68.453,-147.5983,6.3571,-13675.4994
C01674=-1.983,58.291,68.419,-146.3472,-0.2658,-13678.0516
C01675=0.000,58.319,68.442,-146.3576,-0.0000,-13680.0000
C01676=0.000,57.118,70.285,-147.5051,-0.0000,-13680.0000
C01677=1.874,57.094,70.261,-147.4920,0.2427,-13681.8799
C01678=4.398,57.039,70.297,-148.8228,-6.3445,-13684.4091
C01679=7.507,57.930,71.114,-168.0576,-14.9242,-13687.3837
C01680=8.875,61.204,73.167,179.9043,1.8957,-13688.2508
C01681=9.674,66.709,75.971,179.9379,4.0477,-13688.2514
C01682=10.553,73.885,78.794,179.9706,4.8251,-13688.1286
C01683=11.527,81.722,80.892,179.9638,5.2899,-13688.0287
C01684=12.662,88.851,81.904,179.0880,5.0444,-13688.1105
C01685=16.202,94.056,82.431,177.8793,2.4545,-13689.7738
C01686=21.776,96.587,82.857,178.5517,0.5851,-13692.7052
C01687=28.231,95.920,83.283,179.8985,0.0000,-13696.4001
C01688=34.916,93.705,83.562,179.9873,-0.0014,-13700.4362
C01689=41.570,90.949,83.562,179.9872,-0.0004,-13704.5637
C01690=47.863,87.788,83.283,179.8948,-0.0014,-13708.5997
C01691=52.900,83.695,82.857,178.5531,-0.5838,-13712.2952
C01692=55.051,77.964,82.431,177.8795,-2.4557,-13715.2262
C01693=53.873,71.781,81.904,179.0860,-5.0477,-13716.8889
C01694=49.635,65.937,80.892,179.9630,-5.2869,-13716.9711
C01695=44.783,59.707,78.794,179.9688,-4.8309,-13716.8716
C01696=40.330,54.011,75.971,179.9397,-4.0486,-13716.7487
C01697=37.003,49.553,73.167,179.9065,-1.8969,-13716.7500
C01698=35.654,46.271,71.114,-168.0570,14.9247,-13717.6160
C01699=37.223,43.442,70.297,-148.8206,6.3398,-13720.5914
C01700=39.047,41.697,70.261,-147.4931,-0.2438,-13723.1202
C01701=40.388,40.388,70.285,-147.5022,-0.0000,-13725.0000
C01702=41.696,39.047,70.261,-147.4931,0.2442,-13726.8791
C01703=43.443,37.223,70.297,-148.8244,-6.3445,-13729.4092
C01704=46.271,35.654,71.114,-168.0570,-14.9247,-13732.3840
C01705=49.553,37.003,73.167,179.9065,1.8969,-13733.2500
C01706=54.011,40.330,75.971,179.9397,4.0486,-13733.2513
C01707=59.707,44.783,78.794,179.9688,4.8309,-13733.1284
C01708=65.937,49.635,80.892,179.9630,5.2869,-13733.0289
C01709=71.781,53.873,81.904,179.0860,5.0477,-13733.1111
C01710=77.964,55.051,82.431,177.8795,2.4557,-13734.7738
C01711=83.695,52.900,82.857,178.5531,0.5838,-13737.7048
C01712=87.788,47.863,83.283,179.8948,0.0014,-13741.4003
C01713=90.949,41.570,83.562,179.9872,0.0004,-13745.4363
C01714=93.705,34.916,83.562,179.9873,0.0014,-13749.5638
C01715=95.920,28.231,83.283,179.8985,-0.0000,-13753.5999
C01716=96.587,21.776,82.857,178.5517,-0.5851,-13757.2948
C01717=94.056,16.202,82.431,177.8793,-2.4545,-13760.2262
C01718=88.851,12.662,81.904,179.0880,-5.0444,-13761.8895
C01719=81.722,11.527,80.892,179.9638,-5.2899,-13761.9713
C01720=73.885,10.553,78.794,179.9706,-4.8251,-13761.8714
C01721=66.709,9.674,75.971,179.9379,-4.0477,-13761.7486
C01722=61.204,8.875,73.167,179.9043,-1.8957,-13761.7492
C01723=57.930,7.507,71.114,-168.0576,14.9242,-13762.6163
C01724=57.039,4.398,70.297,-148.8228,6.3445,-13765.5909
C01725=57.094,1.874,70.261,-147.4920,-0.2427,-13768.1201
